REGION Network 10: Pulsing temperature and pressure same
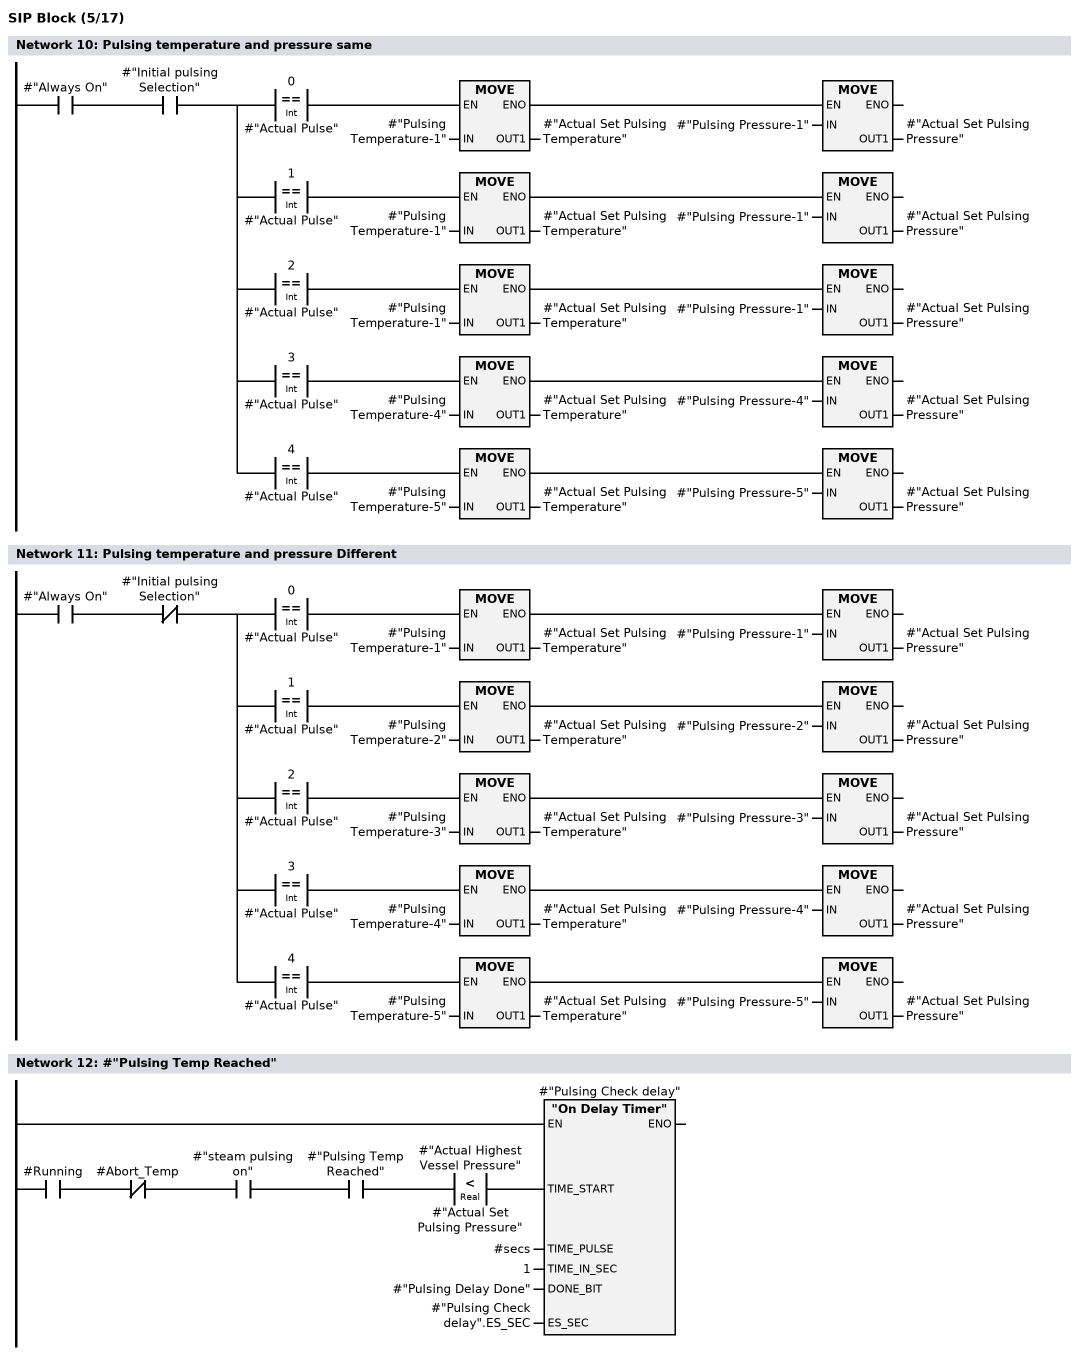
   RUNG wire#powerrail
      Contact( #"Always On" )
      Contact( #"Initial pulsing Selection" )
      wire#w1
      { S7_Templates := "SrcType := Int" } EQ_Contact(in1 := 0, in2 := #"Actual Pulse")
      Move(in := #"Pulsing Temperature-1", out1 => #"Actual Set Pulsing Temperature")
      Move(in := #"Pulsing Pressure-1", out1 => #"Actual Set Pulsing Pressure")
   END_RUNG
   RUNG wire#w1
      { S7_Templates := "SrcType := Int" } EQ_Contact(in1 := 1, in2 := #"Actual Pulse")
      Move(in := #"Pulsing Temperature-1", out1 => #"Actual Set Pulsing Temperature")
      Move(in := #"Pulsing Pressure-1", out1 => #"Actual Set Pulsing Pressure")
   END_RUNG
   RUNG wire#w1
      { S7_Templates := "SrcType := Int" } EQ_Contact(in1 := 2, in2 := #"Actual Pulse")
      Move(in := #"Pulsing Temperature-1", out1 => #"Actual Set Pulsing Temperature")
      Move(in := #"Pulsing Pressure-1", out1 => #"Actual Set Pulsing Pressure")
   END_RUNG
   RUNG wire#w1
      { S7_Templates := "SrcType := Int" } EQ_Contact(in1 := 3, in2 := #"Actual Pulse")
      Move(in := #"Pulsing Temperature-4", out1 => #"Actual Set Pulsing Temperature")
      Move(in := #"Pulsing Pressure-4", out1 => #"Actual Set Pulsing Pressure")
   END_RUNG
   RUNG wire#w1
      { S7_Templates := "SrcType := Int" } EQ_Contact(in1 := 4, in2 := #"Actual Pulse")
      Move(in := #"Pulsing Temperature-5", out1 => #"Actual Set Pulsing Temperature")
      Move(in := #"Pulsing Pressure-5", out1 => #"Actual Set Pulsing Pressure")
   END_RUNG
   // the same network as SCL:
   #_w1 := #"Always On" AND #"Initial pulsing Selection";
   IF #_w1 AND (0 = #"Actual Pulse") THEN
       #"Actual Set Pulsing Temperature" := #"Pulsing Temperature-1";
       #"Actual Set Pulsing Pressure" := #"Pulsing Pressure-1";
   END_IF;
   IF #_w1 AND (1 = #"Actual Pulse") THEN
       #"Actual Set Pulsing Temperature" := #"Pulsing Temperature-1";
       #"Actual Set Pulsing Pressure" := #"Pulsing Pressure-1";
   END_IF;
   IF #_w1 AND (2 = #"Actual Pulse") THEN
       #"Actual Set Pulsing Temperature" := #"Pulsing Temperature-1";
       #"Actual Set Pulsing Pressure" := #"Pulsing Pressure-1";
   END_IF;
   IF #_w1 AND (3 = #"Actual Pulse") THEN
       #"Actual Set Pulsing Temperature" := #"Pulsing Temperature-4";
       #"Actual Set Pulsing Pressure" := #"Pulsing Pressure-4";
   END_IF;
   IF #_w1 AND (4 = #"Actual Pulse") THEN
       #"Actual Set Pulsing Temperature" := #"Pulsing Temperature-5";
       #"Actual Set Pulsing Pressure" := #"Pulsing Pressure-5";
   END_IF;
END_REGION

REGION Network 11: Pulsing temperature and pressure Different
   RUNG wire#powerrail
      Contact( #"Always On" )
      I_Contact( #"Initial pulsing Selection" )
      wire#w1
      { S7_Templates := "SrcType := Int" } EQ_Contact(in1 := 0, in2 := #"Actual Pulse")
      Move(in := #"Pulsing Temperature-1", out1 => #"Actual Set Pulsing Temperature")
      Move(in := #"Pulsing Pressure-1", out1 => #"Actual Set Pulsing Pressure")
   END_RUNG
   RUNG wire#w1
      { S7_Templates := "SrcType := Int" } EQ_Contact(in1 := 1, in2 := #"Actual Pulse")
      Move(in := #"Pulsing Temperature-2", out1 => #"Actual Set Pulsing Temperature")
      Move(in := #"Pulsing Pressure-2", out1 => #"Actual Set Pulsing Pressure")
   END_RUNG
   RUNG wire#w1
      { S7_Templates := "SrcType := Int" } EQ_Contact(in1 := 2, in2 := #"Actual Pulse")
      Move(in := #"Pulsing Temperature-3", out1 => #"Actual Set Pulsing Temperature")
      Move(in := #"Pulsing Pressure-3", out1 => #"Actual Set Pulsing Pressure")
   END_RUNG
   RUNG wire#w1
      { S7_Templates := "SrcType := Int" } EQ_Contact(in1 := 3, in2 := #"Actual Pulse")
      Move(in := #"Pulsing Temperature-4", out1 => #"Actual Set Pulsing Temperature")
      Move(in := #"Pulsing Pressure-4", out1 => #"Actual Set Pulsing Pressure")
   END_RUNG
   RUNG wire#w1
      { S7_Templates := "SrcType := Int" } EQ_Contact(in1 := 4, in2 := #"Actual Pulse")
      Move(in := #"Pulsing Temperature-5", out1 => #"Actual Set Pulsing Temperature")
      Move(in := #"Pulsing Pressure-5", out1 => #"Actual Set Pulsing Pressure")
   END_RUNG
   // the same network as SCL:
   #_w1 := #"Always On" AND NOT #"Initial pulsing Selection";
   IF #_w1 AND (0 = #"Actual Pulse") THEN
       #"Actual Set Pulsing Temperature" := #"Pulsing Temperature-1";
       #"Actual Set Pulsing Pressure" := #"Pulsing Pressure-1";
   END_IF;
   IF #_w1 AND (1 = #"Actual Pulse") THEN
       #"Actual Set Pulsing Temperature" := #"Pulsing Temperature-2";
       #"Actual Set Pulsing Pressure" := #"Pulsing Pressure-2";
   END_IF;
   IF #_w1 AND (2 = #"Actual Pulse") THEN
       #"Actual Set Pulsing Temperature" := #"Pulsing Temperature-3";
       #"Actual Set Pulsing Pressure" := #"Pulsing Pressure-3";
   END_IF;
   IF #_w1 AND (3 = #"Actual Pulse") THEN
       #"Actual Set Pulsing Temperature" := #"Pulsing Temperature-4";
       #"Actual Set Pulsing Pressure" := #"Pulsing Pressure-4";
   END_IF;
   IF #_w1 AND (4 = #"Actual Pulse") THEN
       #"Actual Set Pulsing Temperature" := #"Pulsing Temperature-5";
       #"Actual Set Pulsing Pressure" := #"Pulsing Pressure-5";
   END_IF;
END_REGION

REGION Network 12: #"Pulsing Temp Reached"
   RUNG wire#powerrail
      #"Pulsing Check delay"(TIME_START := wire#w1, TIME_PULSE := #secs, TIME_IN_SEC := 1, DONE_BIT := #"Pulsing Delay Done", ES_SEC := #"Pulsing Check delay".ES_SEC)
   END_RUNG
   RUNG wire#powerrail
      Contact( #Running )
      I_Contact( #Abort_Temp )
      Contact( #"steam pulsing on" )
      Contact( #"Pulsing Temp Reached" )
      { S7_Templates := "SrcType := Real" } LT_Contact(in1 := #"Actual Highest Vessel Pressure", in2 := #"Actual Set Pulsing Pressure")
   END_RUNG wire#w1
   // the same network as SCL:
   #"Pulsing Check delay"(TIME_START := #Running AND NOT #Abort_Temp AND #"steam pulsing on" AND #"Pulsing Temp Reached" AND (#"Actual Highest Vessel Pressure" < #"Actual Set Pulsing Pressure"),   // "On Delay Timer"
                          TIME_PULSE := #secs,
                          TIME_IN_SEC := 1,
                          DONE_BIT := #"Pulsing Delay Done",
                          ES_SEC := #"Pulsing Check delay".ES_SEC);
END_REGION

REGION Network 13: #"Pulsing Temp Reached"
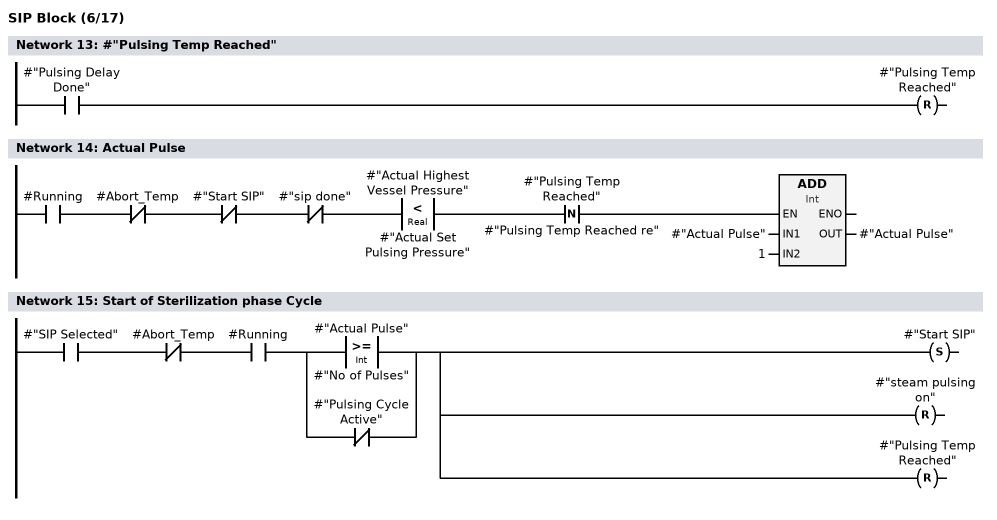
   RUNG wire#powerrail
      Contact( #"Pulsing Delay Done" )
      R_Coil( #"Pulsing Temp Reached" )
   END_RUNG
   // the same network as SCL:
   IF #"Pulsing Delay Done" THEN #"Pulsing Temp Reached" := FALSE; END_IF;
END_REGION

REGION Network 14: Actual Pulse
   RUNG wire#powerrail
      Contact( #Running )
      I_Contact( #Abort_Temp )
      I_Contact( #"Start SIP" )
      I_Contact( #"sip done" )
      { S7_Templates := "SrcType := Real" } LT_Contact(in1 := #"Actual Highest Vessel Pressure", in2 := #"Actual Set Pulsing Pressure")
      N_Contact(operand := #"Pulsing Temp Reached", bit := #"Pulsing Temp Reached re")
      { S7_Templates := "SrcType := Int"; S7_GenerateENO := "TRUE" } Add(in1 := #"Actual Pulse", in2 := 1, out => #"Actual Pulse")
   END_RUNG
   // the same network as SCL:
   #_w1 := #Running AND NOT #Abort_Temp AND NOT #"Start SIP" AND NOT #"sip done" AND (#"Actual Highest Vessel Pressure" < #"Actual Set Pulsing Pressure") AND NOT #"Pulsing Temp Reached" AND #"Pulsing Temp Reached re";   // falling edge of #"Pulsing Temp Reached"
   #"Pulsing Temp Reached re" := #"Pulsing Temp Reached";
   IF #_w1 THEN #"Actual Pulse" := #"Actual Pulse" + 1; END_IF;
END_REGION

REGION Network 15: Start of Sterilization phase Cycle
   RUNG wire#powerrail
      Contact( #"SIP Selected" )
      I_Contact( #Abort_Temp )
      Contact( #Running )
      wire#w1
      { S7_Templates := "SrcType := Int" } GE_Contact(in1 := #"Actual Pulse", in2 := #"No of Pulses")
      wire#w2
      S_Coil( #"Start SIP" )
   END_RUNG
   RUNG wire#w1
      I_Contact( #"Pulsing Cycle Active" )
   END_RUNG wire#w2
   RUNG wire#w2
      R_Coil( #"steam pulsing on" )
   END_RUNG
   RUNG wire#w2
      R_Coil( #"Pulsing Temp Reached" )
   END_RUNG
   // the same network as SCL:
   IF #"SIP Selected" AND NOT #Abort_Temp AND #Running AND ((#"Actual Pulse" >= #"No of Pulses") OR NOT #"Pulsing Cycle Active") THEN
       #"Start SIP" := TRUE;
       #"steam pulsing on" := FALSE;
       #"Pulsing Temp Reached" := FALSE;
   END_IF;
END_REGION

REGION Network 16: SIP Logic
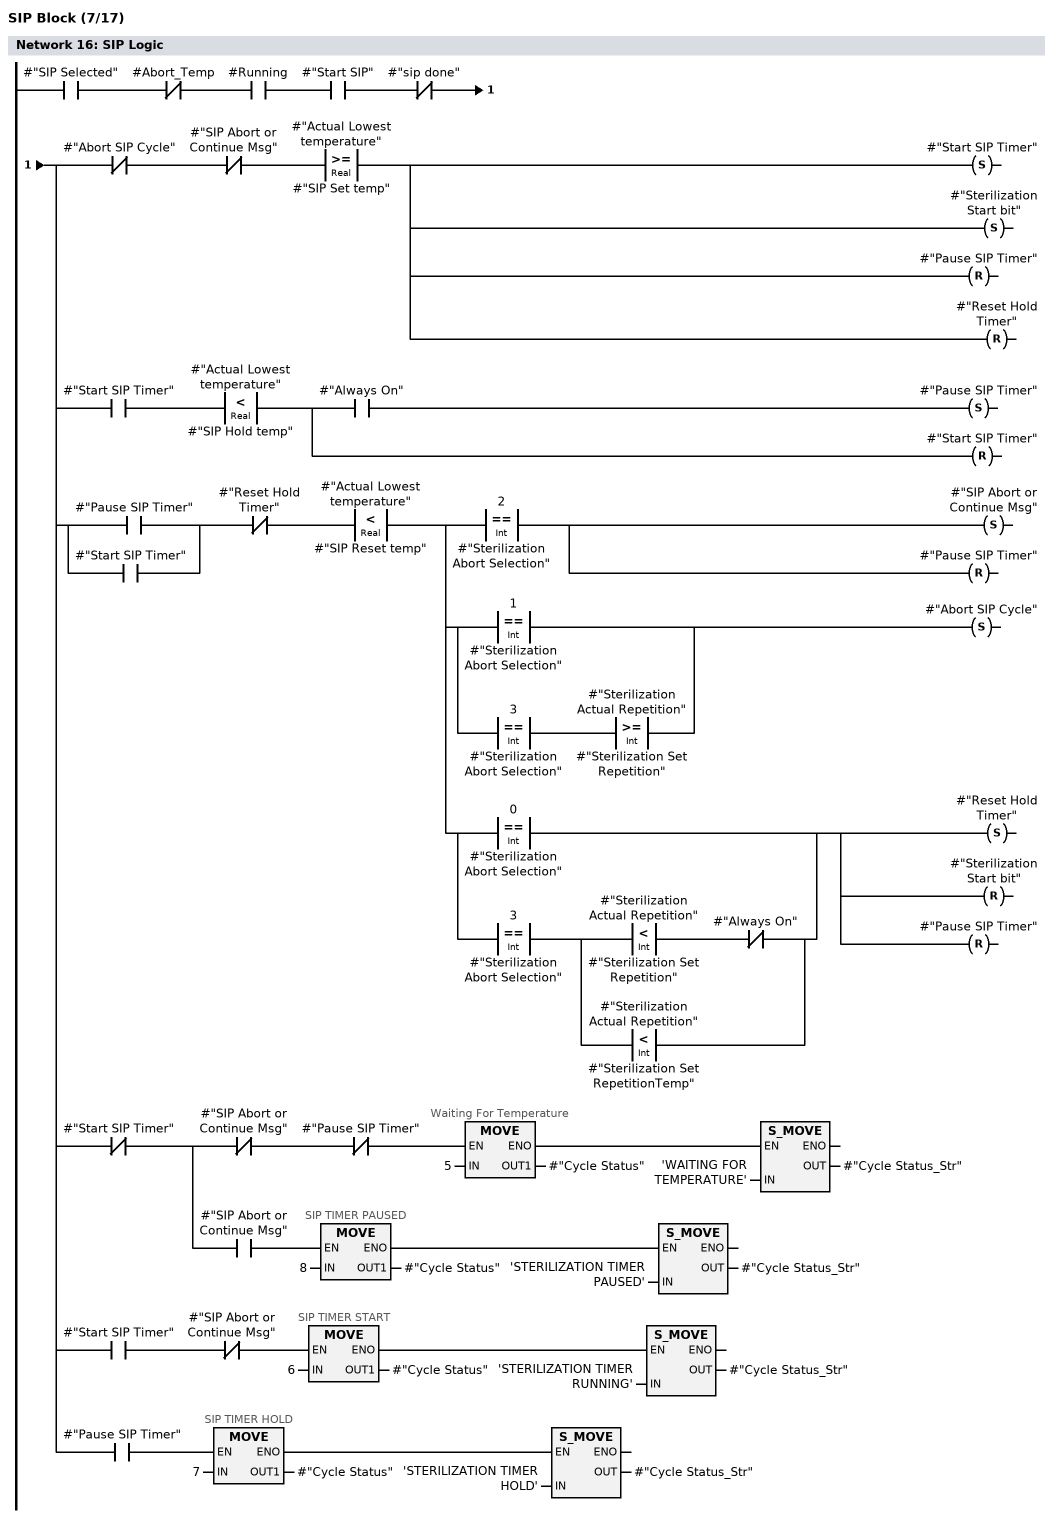
   RUNG wire#powerrail
      Contact( #"SIP Selected" )
      I_Contact( #Abort_Temp )
      Contact( #Running )
      Contact( #"Start SIP" )
      I_Contact( #"sip done" )
      wire#w1
      I_Contact( #"Abort SIP Cycle" )
      I_Contact( #"SIP Abort or Continue Msg" )
      { S7_Templates := "SrcType := Real" } GE_Contact(in1 := #"Actual Lowest temperature", in2 := #"SIP Set temp")
      wire#w2
      S_Coil( #"Start SIP Timer" )
   END_RUNG
   RUNG wire#w2
      S_Coil( #"Sterilization Start bit" )
   END_RUNG
   RUNG wire#w2
      R_Coil( #"Pause SIP Timer" )
   END_RUNG
   RUNG wire#w2
      R_Coil( #"Reset Hold Timer" )
   END_RUNG
   RUNG wire#w1
      Contact( #"Start SIP Timer" )
      { S7_Templates := "SrcType := Real" } LT_Contact(in1 := #"Actual Lowest temperature", in2 := #"SIP Hold temp")
      wire#w3
      Contact( #"Always On" )
      S_Coil( #"Pause SIP Timer" )
   END_RUNG
   RUNG wire#w3
      R_Coil( #"Start SIP Timer" )
   END_RUNG
   RUNG wire#w1
      Contact( #"Pause SIP Timer" )
      wire#w4
      I_Contact( #"Reset Hold Timer" )
      { S7_Templates := "SrcType := Real" } LT_Contact(in1 := #"Actual Lowest temperature", in2 := #"SIP Reset temp")
      wire#w5
      { S7_Templates := "SrcType := Int" } EQ_Contact(in1 := 2, in2 := #"Sterilization Abort Selection")
      wire#w6
      S_Coil( #"SIP Abort or Continue Msg" )
   END_RUNG
   RUNG wire#w1
      Contact( #"Start SIP Timer" )
   END_RUNG wire#w4
   RUNG wire#w6
      R_Coil( #"Pause SIP Timer" )
   END_RUNG
   RUNG wire#w5
      { S7_Templates := "SrcType := Int" } EQ_Contact(in1 := 1, in2 := #"Sterilization Abort Selection")
      wire#w7
      S_Coil( #"Abort SIP Cycle" )
   END_RUNG
   RUNG wire#w5
      { S7_Templates := "SrcType := Int" } EQ_Contact(in1 := 3, in2 := #"Sterilization Abort Selection")
      { S7_Templates := "SrcType := Int" } GE_Contact(in1 := #"Sterilization Actual Repetition", in2 := #"Sterilization Set Repetition")
   END_RUNG wire#w7
   RUNG wire#w5
      { S7_Templates := "SrcType := Int" } EQ_Contact(in1 := 0, in2 := #"Sterilization Abort Selection")
      wire#w8
      S_Coil( #"Reset Hold Timer" )
   END_RUNG
   RUNG wire#w5
      { S7_Templates := "SrcType := Int" } EQ_Contact(in1 := 3, in2 := #"Sterilization Abort Selection")
      wire#w9
      { S7_Templates := "SrcType := Int" } LT_Contact(in1 := #"Sterilization Actual Repetition", in2 := #"Sterilization Set Repetition")
      I_Contact( #"Always On" )
   END_RUNG wire#w8
   RUNG wire#w9
      { S7_Templates := "SrcType := Int" } LT_Contact(in1 := #"Sterilization Actual Repetition", in2 := #"Sterilization Set RepetitionTemp")
   END_RUNG wire#w8
   RUNG wire#w8
      R_Coil( #"Sterilization Start bit" )
   END_RUNG
   RUNG wire#w8
      R_Coil( #"Pause SIP Timer" )
   END_RUNG
   RUNG wire#w1
      I_Contact( #"Start SIP Timer" )
      wire#w10
      I_Contact( #"SIP Abort or Continue Msg" )
      I_Contact( #"Pause SIP Timer" )
      { S7_GenerateENO := "TRUE" } Move(in := 5, out1 => #"Cycle Status")   // Waiting For Temperature
      S_Move(in := 'WAITING FOR TEMPERATURE', out => #"Cycle Status_Str")
   END_RUNG
   RUNG wire#w10
      Contact( #"SIP Abort or Continue Msg" )
      { S7_GenerateENO := "TRUE" } Move(in := 8, out1 => #"Cycle Status")   // SIP TIMER PAUSED
      S_Move(in := 'STERILIZATION TIMER PAUSED', out => #"Cycle Status_Str")
   END_RUNG
   RUNG wire#w1
      Contact( #"Start SIP Timer" )
      I_Contact( #"SIP Abort or Continue Msg" )
      { S7_GenerateENO := "TRUE" } Move(in := 6, out1 => #"Cycle Status")   // SIP TIMER START
      S_Move(in := 'STERILIZATION TIMER RUNNING', out => #"Cycle Status_Str")
   END_RUNG
   RUNG wire#w1
      Contact( #"Pause SIP Timer" )
      { S7_GenerateENO := "TRUE" } Move(in := 7, out1 => #"Cycle Status")   // SIP TIMER HOLD
      S_Move(in := 'STERILIZATION TIMER HOLD', out => #"Cycle Status_Str")
   END_RUNG
   // the same network as SCL:
   // ENO of a box is taken as its EN; it also drops when the box reports an error
   #_w1 := #"SIP Selected" AND NOT #Abort_Temp AND #Running AND #"Start SIP" AND NOT #"sip done";
   IF #_w1 AND NOT #"Abort SIP Cycle" AND NOT #"SIP Abort or Continue Msg" AND (#"Actual Lowest temperature" >= #"SIP Set temp") THEN
       #"Start SIP Timer" := TRUE;
       #"Sterilization Start bit" := TRUE;
       #"Pause SIP Timer" := FALSE;
       #"Reset Hold Timer" := FALSE;
   END_IF;
   #_w2 := #_w1 AND #"Start SIP Timer" AND (#"Actual Lowest temperature" < #"SIP Hold temp");
   IF #_w2 AND #"Always On" THEN #"Pause SIP Timer" := TRUE; END_IF;
   IF #_w2 THEN #"Start SIP Timer" := FALSE; END_IF;
   #_w3 := #_w1 AND (#"Pause SIP Timer" OR #"Start SIP Timer") AND NOT #"Reset Hold Timer" AND (#"Actual Lowest temperature" < #"SIP Reset temp");
   IF #_w3 AND (2 = #"Sterilization Abort Selection") THEN
       #"SIP Abort or Continue Msg" := TRUE;
       #"Pause SIP Timer" := FALSE;
   END_IF;
   IF #_w3 AND ((1 = #"Sterilization Abort Selection") OR ((3 = #"Sterilization Abort Selection") AND (#"Sterilization Actual Repetition" >= #"Sterilization Set Repetition"))) THEN
       #"Abort SIP Cycle" := TRUE;
   END_IF;
   IF #_w3 AND ((0 = #"Sterilization Abort Selection") OR ((3 = #"Sterilization Abort Selection") AND (((#"Sterilization Actual Repetition" < #"Sterilization Set Repetition") AND NOT #"Always On") OR (#"Sterilization Actual Repetition" < #"Sterilization Set RepetitionTemp")))) THEN
       #"Reset Hold Timer" := TRUE;
       #"Sterilization Start bit" := FALSE;
       #"Pause SIP Timer" := FALSE;
   END_IF;
   #_w4 := #_w1 AND NOT #"Start SIP Timer";
   IF #_w4 AND NOT #"SIP Abort or Continue Msg" AND NOT #"Pause SIP Timer" THEN
       #"Cycle Status" := 5;   // Waiting For Temperature
       #"Cycle Status_Str" := 'WAITING FOR TEMPERATURE';
   END_IF;
   IF #_w4 AND #"SIP Abort or Continue Msg" THEN
       #"Cycle Status" := 8;   // SIP TIMER PAUSED
       #"Cycle Status_Str" := 'STERILIZATION TIMER PAUSED';
   END_IF;
   IF #_w1 AND #"Start SIP Timer" AND NOT #"SIP Abort or Continue Msg" THEN
       #"Cycle Status" := 6;   // SIP TIMER START
       #"Cycle Status_Str" := 'STERILIZATION TIMER RUNNING';
   END_IF;
   IF #_w1 AND #"Pause SIP Timer" THEN
       #"Cycle Status" := 7;   // SIP TIMER HOLD
       #"Cycle Status_Str" := 'STERILIZATION TIMER HOLD';
   END_IF;
END_REGION

REGION Network 17: Selection 2 :Abort msg conditions
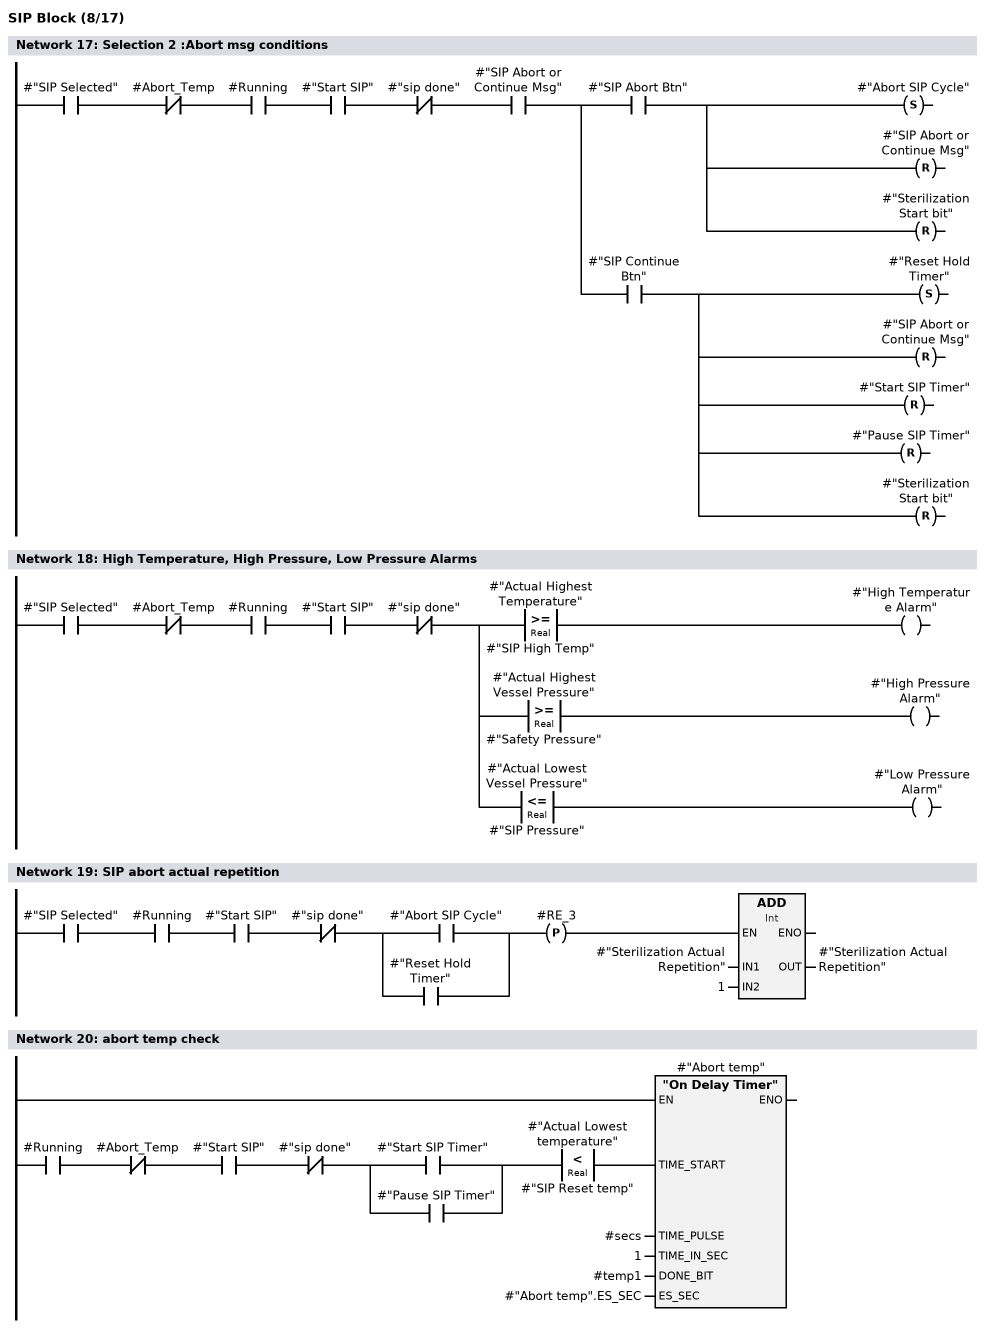
   RUNG wire#powerrail
      Contact( #"SIP Selected" )
      I_Contact( #Abort_Temp )
      Contact( #Running )
      Contact( #"Start SIP" )
      I_Contact( #"sip done" )
      Contact( #"SIP Abort or Continue Msg" )
      wire#w1
      Contact( #"SIP Abort Btn" )
      wire#w2
      S_Coil( #"Abort SIP Cycle" )
   END_RUNG
   RUNG wire#w2
      R_Coil( #"SIP Abort or Continue Msg" )
   END_RUNG
   RUNG wire#w2
      R_Coil( #"Sterilization Start bit" )
   END_RUNG
   RUNG wire#w1
      Contact( #"SIP Continue Btn" )
      wire#w3
      S_Coil( #"Reset Hold Timer" )
   END_RUNG
   RUNG wire#w3
      R_Coil( #"SIP Abort or Continue Msg" )
   END_RUNG
   RUNG wire#w3
      R_Coil( #"Start SIP Timer" )
   END_RUNG
   RUNG wire#w3
      R_Coil( #"Pause SIP Timer" )
   END_RUNG
   RUNG wire#w3
      R_Coil( #"Sterilization Start bit" )
   END_RUNG
   // the same network as SCL:
   #_w1 := #"SIP Selected" AND NOT #Abort_Temp AND #Running AND #"Start SIP" AND NOT #"sip done" AND #"SIP Abort or Continue Msg";
   IF #_w1 AND #"SIP Abort Btn" THEN
       #"Abort SIP Cycle" := TRUE;
       #"SIP Abort or Continue Msg" := FALSE;
       #"Sterilization Start bit" := FALSE;
   END_IF;
   IF #_w1 AND #"SIP Continue Btn" THEN
       #"Reset Hold Timer" := TRUE;
       #"SIP Abort or Continue Msg" := FALSE;
       #"Start SIP Timer" := FALSE;
       #"Pause SIP Timer" := FALSE;
       #"Sterilization Start bit" := FALSE;
   END_IF;
END_REGION

REGION Network 18: High Temperature, High Pressure, Low Pressure Alarms
   RUNG wire#powerrail
      Contact( #"SIP Selected" )
      I_Contact( #Abort_Temp )
      Contact( #Running )
      Contact( #"Start SIP" )
      I_Contact( #"sip done" )
      wire#w1
      { S7_Templates := "SrcType := Real" } GE_Contact(in1 := #"Actual Highest Temperature", in2 := #"SIP High Temp")
      Coil( #"High Temperature Alarm" )
   END_RUNG
   RUNG wire#w1
      { S7_Templates := "SrcType := Real" } GE_Contact(in1 := #"Actual Highest Vessel Pressure", in2 := #"Safety Pressure")
      Coil( #"High Pressure Alarm" )
   END_RUNG
   RUNG wire#w1
      { S7_Templates := "SrcType := Real" } LE_Contact(in1 := #"Actual Lowest Vessel Pressure", in2 := #"SIP Pressure")
      Coil( #"Low Pressure Alarm" )
   END_RUNG
   // the same network as SCL:
   #_w1 := #"SIP Selected" AND NOT #Abort_Temp AND #Running AND #"Start SIP" AND NOT #"sip done";
   #"High Temperature Alarm" := #_w1 AND (#"Actual Highest Temperature" >= #"SIP High Temp");
   #"High Pressure Alarm" := #_w1 AND (#"Actual Highest Vessel Pressure" >= #"Safety Pressure");
   #"Low Pressure Alarm" := #_w1 AND (#"Actual Lowest Vessel Pressure" <= #"SIP Pressure");
END_REGION

REGION Network 19: SIP abort actual repetition
   RUNG wire#powerrail
      Contact( #"SIP Selected" )
      Contact( #Running )
      Contact( #"Start SIP" )
      I_Contact( #"sip done" )
      wire#w1
      Contact( #"Abort SIP Cycle" )
      wire#w2
      P_Trig( #RE_3 )
      { S7_Templates := "SrcType := Int" } Add(in1 := #"Sterilization Actual Repetition", in2 := 1, out => #"Sterilization Actual Repetition")
   END_RUNG
   RUNG wire#w1
      Contact( #"Reset Hold Timer" )
   END_RUNG wire#w2
   // the same network as SCL:
   #_w1 := #"SIP Selected" AND #Running AND #"Start SIP" AND NOT #"sip done" AND (#"Abort SIP Cycle" OR #"Reset Hold Timer");
   #_w2 := #_w1 AND NOT #RE_3;   // rising edge
   #RE_3 := #_w1;
   IF #_w2 THEN #"Sterilization Actual Repetition" := #"Sterilization Actual Repetition" + 1; END_IF;
END_REGION

REGION Network 20: abort temp check
   RUNG wire#powerrail
      #"Abort temp"(TIME_START := wire#w3, TIME_PULSE := #secs, TIME_IN_SEC := 1, DONE_BIT := #temp1, ES_SEC := #"Abort temp".ES_SEC)
   END_RUNG
   RUNG wire#powerrail
      Contact( #Running )
      I_Contact( #Abort_Temp )
      Contact( #"Start SIP" )
      I_Contact( #"sip done" )
      wire#w1
      Contact( #"Start SIP Timer" )
      wire#w2
      { S7_Templates := "SrcType := Real" } LT_Contact(in1 := #"Actual Lowest temperature", in2 := #"SIP Reset temp")
   END_RUNG wire#w3
   RUNG wire#w1
      Contact( #"Pause SIP Timer" )
   END_RUNG wire#w2
   // the same network as SCL:
   #"Abort temp"(TIME_START := #Running AND NOT #Abort_Temp AND #"Start SIP" AND NOT #"sip done" AND (#"Start SIP Timer" OR #"Pause SIP Timer") AND (#"Actual Lowest temperature" < #"SIP Reset temp"),   // "On Delay Timer"
                 TIME_PULSE := #secs,
                 TIME_IN_SEC := 1,
                 DONE_BIT := #temp1,
                 ES_SEC := #"Abort temp".ES_SEC);
END_REGION

REGION Network 21: sip hold timer
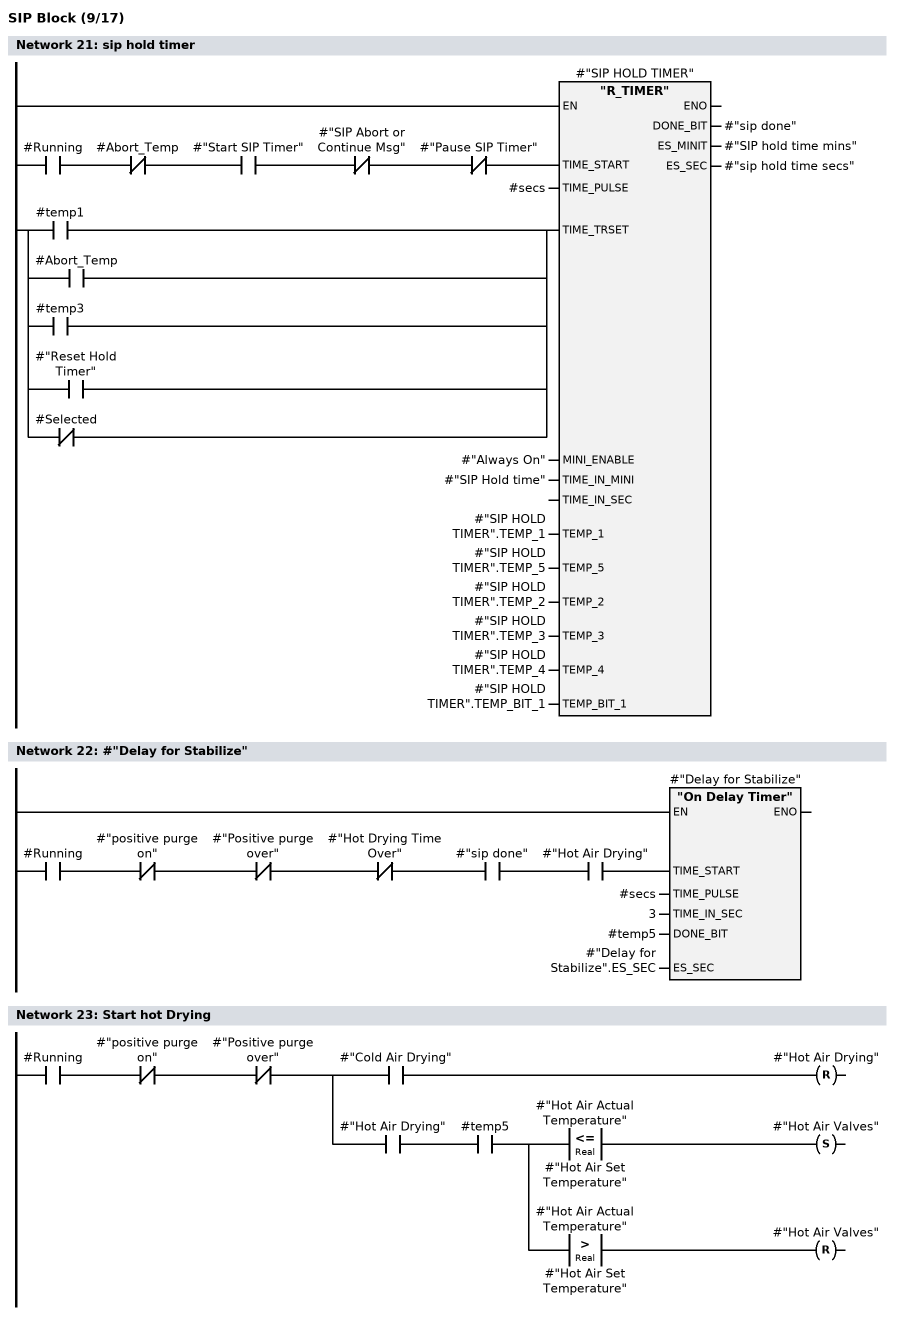
   RUNG wire#powerrail
      #"SIP HOLD TIMER"(TIME_START := wire#w1, TIME_TRSET := wire#w2, TIME_PULSE := #secs, MINI_ENABLE := #"Always On", TIME_IN_MINI := #"SIP Hold time", TIME_IN_SEC :=, TEMP_1 := #"SIP HOLD TIMER".TEMP_1, TEMP_5 := #"SIP HOLD TIMER".TEMP_5, TEMP_2 := #"SIP HOLD TIMER".TEMP_2, TEMP_3 := #"SIP HOLD TIMER".TEMP_3, TEMP_4 := #"SIP HOLD TIMER".TEMP_4, TEMP_BIT_1 := #"SIP HOLD TIMER".TEMP_BIT_1, DONE_BIT => #"sip done", ES_MINIT => #"SIP hold time mins", ES_SEC => #"sip hold time secs")
   END_RUNG
   RUNG wire#powerrail
      Contact( #Running )
      I_Contact( #Abort_Temp )
      Contact( #"Start SIP Timer" )
      I_Contact( #"SIP Abort or Continue Msg" )
      I_Contact( #"Pause SIP Timer" )
   END_RUNG wire#w1
   RUNG wire#powerrail
      Contact( #temp1 )
   END_RUNG wire#w2
   RUNG wire#powerrail
      Contact( #Abort_Temp )
   END_RUNG wire#w2
   RUNG wire#powerrail
      Contact( #temp3 )
   END_RUNG wire#w2
   RUNG wire#powerrail
      Contact( #"Reset Hold Timer" )
   END_RUNG wire#w2
   RUNG wire#powerrail
      I_Contact( #Selected )
   END_RUNG wire#w2
   // the same network as SCL:
   #"SIP HOLD TIMER"(TIME_START := #Running AND NOT #Abort_Temp AND #"Start SIP Timer" AND NOT #"SIP Abort or Continue Msg" AND NOT #"Pause SIP Timer",   // "R_TIMER"
                     TIME_PULSE := #secs,
                     TIME_TRSET := #temp1 OR #Abort_Temp OR #temp3 OR #"Reset Hold Timer" OR NOT #Selected,
                     MINI_ENABLE := #"Always On",
                     TIME_IN_MINI := #"SIP Hold time",
                     TEMP_1 := #"SIP HOLD TIMER".TEMP_1,
                     TEMP_5 := #"SIP HOLD TIMER".TEMP_5,
                     TEMP_2 := #"SIP HOLD TIMER".TEMP_2,
                     TEMP_3 := #"SIP HOLD TIMER".TEMP_3,
                     TEMP_4 := #"SIP HOLD TIMER".TEMP_4,
                     TEMP_BIT_1 := #"SIP HOLD TIMER".TEMP_BIT_1,
                     DONE_BIT => #"sip done",
                     ES_MINIT => #"SIP hold time mins",
                     ES_SEC => #"sip hold time secs");
END_REGION

REGION Network 22: #"Delay for Stabilize"
   RUNG wire#powerrail
      #"Delay for Stabilize"(TIME_START := wire#w1, TIME_PULSE := #secs, TIME_IN_SEC := 3, DONE_BIT := #temp5, ES_SEC := #"Delay for Stabilize".ES_SEC)
   END_RUNG
   RUNG wire#powerrail
      Contact( #Running )
      I_Contact( #"positive purge on" )
      I_Contact( #"Positive purge over" )
      I_Contact( #"Hot Drying Time Over" )
      Contact( #"sip done" )
      Contact( #"Hot Air Drying" )
   END_RUNG wire#w1
   // the same network as SCL:
   #"Delay for Stabilize"(TIME_START := #Running AND NOT #"positive purge on" AND NOT #"Positive purge over" AND NOT #"Hot Drying Time Over" AND #"sip done" AND #"Hot Air Drying",   // "On Delay Timer"
                          TIME_PULSE := #secs,
                          TIME_IN_SEC := 3,
                          DONE_BIT := #temp5,
                          ES_SEC := #"Delay for Stabilize".ES_SEC);
END_REGION

REGION Network 23: Start hot Drying
   RUNG wire#powerrail
      Contact( #Running )
      I_Contact( #"positive purge on" )
      I_Contact( #"Positive purge over" )
      wire#w1
      Contact( #"Cold Air Drying" )
      R_Coil( #"Hot Air Drying" )
   END_RUNG
   RUNG wire#w1
      Contact( #"Hot Air Drying" )
      Contact( #temp5 )
      wire#w2
      { S7_Templates := "SrcType := Real" } LE_Contact(in1 := #"Hot Air Actual Temperature", in2 := #"Hot Air Set Temperature")
      S_Coil( #"Hot Air Valves" )
   END_RUNG
   RUNG wire#w2
      { S7_Templates := "SrcType := Real" } GT_Contact(in1 := #"Hot Air Actual Temperature", in2 := #"Hot Air Set Temperature")
      R_Coil( #"Hot Air Valves" )
   END_RUNG
   // the same network as SCL:
   #_w1 := #Running AND NOT #"positive purge on" AND NOT #"Positive purge over";
   IF #_w1 AND #"Cold Air Drying" THEN #"Hot Air Drying" := FALSE; END_IF;
   #_w2 := #_w1 AND #"Hot Air Drying" AND #temp5;
   IF #_w2 AND (#"Hot Air Actual Temperature" <= #"Hot Air Set Temperature") THEN
       #"Hot Air Valves" := TRUE;
   END_IF;
   IF #_w2 AND (#"Hot Air Actual Temperature" > #"Hot Air Set Temperature") THEN
       #"Hot Air Valves" := FALSE;
   END_IF;
END_REGION

REGION Network 24: Hot Air Drying #"Actual Highest Vessel Pressure"
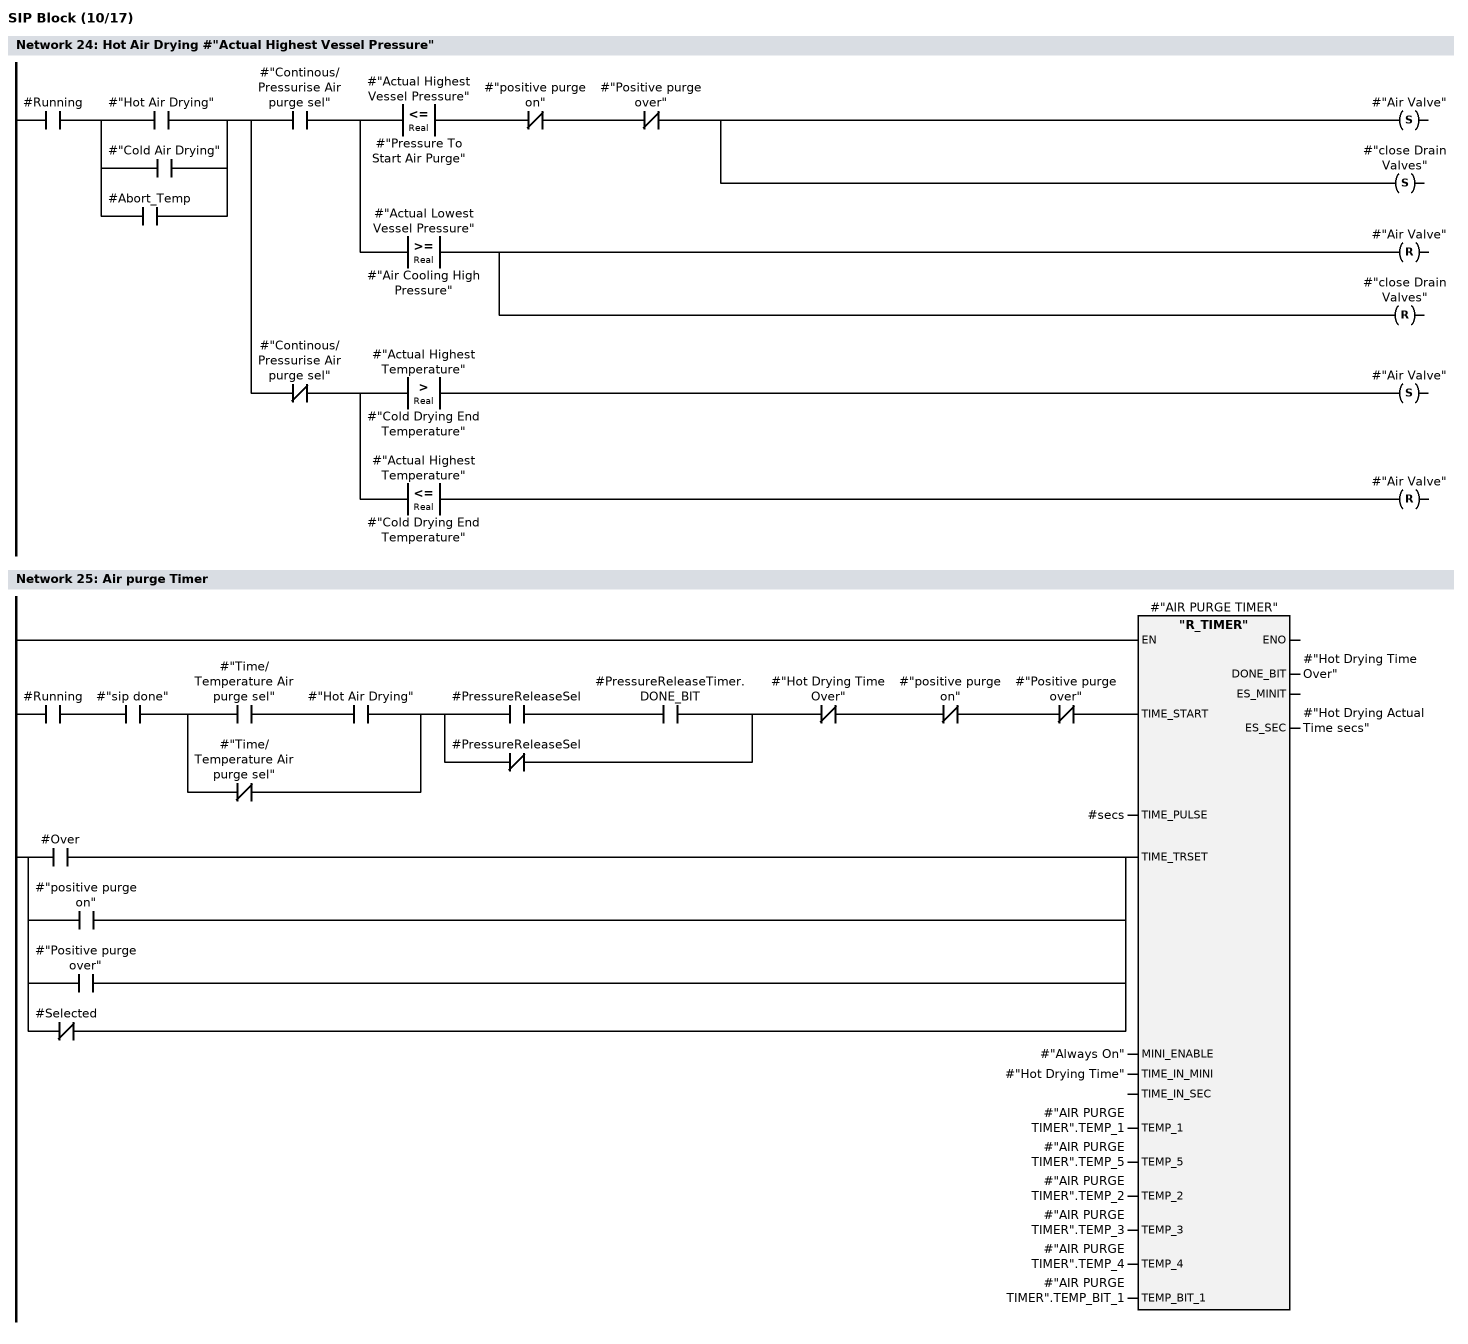
   RUNG wire#powerrail
      Contact( #Running )
      wire#w1
      Contact( #"Hot Air Drying" )
      wire#w2
      Contact( #"Continous/Pressurise Air purge sel" )
      wire#w3
      { S7_Templates := "SrcType := Real" } LE_Contact(in1 := #"Actual Highest Vessel Pressure", in2 := #"Pressure To Start Air Purge")
      I_Contact( #"positive purge on" )
      I_Contact( #"Positive purge over" )
      wire#w4
      S_Coil( #"Air Valve" )
   END_RUNG
   RUNG wire#w1
      Contact( #"Cold Air Drying" )
   END_RUNG wire#w2
   RUNG wire#w1
      Contact( #Abort_Temp )
   END_RUNG wire#w2
   RUNG wire#w4
      S_Coil( #"close Drain Valves" )
   END_RUNG
   RUNG wire#w3
      { S7_Templates := "SrcType := Real" } GE_Contact(in1 := #"Actual Lowest Vessel Pressure", in2 := #"Air Cooling High Pressure")
      wire#w5
      R_Coil( #"Air Valve" )
   END_RUNG
   RUNG wire#w5
      R_Coil( #"close Drain Valves" )
   END_RUNG
   RUNG wire#w2
      I_Contact( #"Continous/Pressurise Air purge sel" )
      wire#w6
      { S7_Templates := "SrcType := Real" } GT_Contact(in1 := #"Actual Highest Temperature", in2 := #"Cold Drying End Temperature")
      S_Coil( #"Air Valve" )
   END_RUNG
   RUNG wire#w6
      { S7_Templates := "SrcType := Real" } LE_Contact(in1 := #"Actual Highest Temperature", in2 := #"Cold Drying End Temperature")
      R_Coil( #"Air Valve" )
   END_RUNG
   // the same network as SCL:
   #_w1 := #Running AND (#"Hot Air Drying" OR #"Cold Air Drying" OR #Abort_Temp);
   #_w2 := #_w1 AND #"Continous/Pressurise Air purge sel";
   IF #_w2 AND (#"Actual Highest Vessel Pressure" <= #"Pressure To Start Air Purge") AND NOT #"positive purge on" AND NOT #"Positive purge over" THEN
       #"Air Valve" := TRUE;
       #"close Drain Valves" := TRUE;
   END_IF;
   IF #_w2 AND (#"Actual Lowest Vessel Pressure" >= #"Air Cooling High Pressure") THEN
       #"Air Valve" := FALSE;
       #"close Drain Valves" := FALSE;
   END_IF;
   #_w3 := #_w1 AND NOT #"Continous/Pressurise Air purge sel";
   IF #_w3 AND (#"Actual Highest Temperature" > #"Cold Drying End Temperature") THEN
       #"Air Valve" := TRUE;
   END_IF;
   IF #_w3 AND (#"Actual Highest Temperature" <= #"Cold Drying End Temperature") THEN
       #"Air Valve" := FALSE;
   END_IF;
END_REGION

REGION Network 25: Air purge Timer
   RUNG wire#powerrail
      #"AIR PURGE TIMER"(TIME_START := wire#w4, TIME_TRSET := wire#w5, TIME_PULSE := #secs, MINI_ENABLE := #"Always On", TIME_IN_MINI := #"Hot Drying Time", TIME_IN_SEC :=, TEMP_1 := #"AIR PURGE TIMER".TEMP_1, TEMP_5 := #"AIR PURGE TIMER".TEMP_5, TEMP_2 := #"AIR PURGE TIMER".TEMP_2, TEMP_3 := #"AIR PURGE TIMER".TEMP_3, TEMP_4 := #"AIR PURGE TIMER".TEMP_4, TEMP_BIT_1 := #"AIR PURGE TIMER".TEMP_BIT_1, DONE_BIT => #"Hot Drying Time Over", ES_MINIT =>, ES_SEC => #"Hot Drying Actual Time secs")
   END_RUNG
   RUNG wire#powerrail
      Contact( #Running )
      Contact( #"sip done" )
      wire#w1
      Contact( #"Time/Temperature Air purge sel" )
      Contact( #"Hot Air Drying" )
      wire#w2
      Contact( #PressureReleaseSel )
      Contact( #PressureReleaseTimer.DONE_BIT )
      wire#w3
      I_Contact( #"Hot Drying Time Over" )
      I_Contact( #"positive purge on" )
      I_Contact( #"Positive purge over" )
   END_RUNG wire#w4
   RUNG wire#w1
      I_Contact( #"Time/Temperature Air purge sel" )
   END_RUNG wire#w2
   RUNG wire#w2
      I_Contact( #PressureReleaseSel )
   END_RUNG wire#w3
   RUNG wire#powerrail
      Contact( #Over )
   END_RUNG wire#w5
   RUNG wire#powerrail
      Contact( #"positive purge on" )
   END_RUNG wire#w5
   RUNG wire#powerrail
      Contact( #"Positive purge over" )
   END_RUNG wire#w5
   RUNG wire#powerrail
      I_Contact( #Selected )
   END_RUNG wire#w5
   // the same network as SCL:
   #"AIR PURGE TIMER"(TIME_START := #Running AND #"sip done" AND ((#"Time/Temperature Air purge sel" AND #"Hot Air Drying") OR NOT #"Time/Temperature Air purge sel") AND ((#PressureReleaseSel AND #PressureReleaseTimer.DONE_BIT) OR NOT #PressureReleaseSel) AND NOT #"Hot Drying Time Over" AND NOT #"positive purge on" AND NOT #"Positive purge over",   // "R_TIMER"
                      TIME_PULSE := #secs,
                      TIME_TRSET := #Over OR #"positive purge on" OR #"Positive purge over" OR NOT #Selected,
                      MINI_ENABLE := #"Always On",
                      TIME_IN_MINI := #"Hot Drying Time",
                      TEMP_1 := #"AIR PURGE TIMER".TEMP_1,
                      TEMP_5 := #"AIR PURGE TIMER".TEMP_5,
                      TEMP_2 := #"AIR PURGE TIMER".TEMP_2,
                      TEMP_3 := #"AIR PURGE TIMER".TEMP_3,
                      TEMP_4 := #"AIR PURGE TIMER".TEMP_4,
                      TEMP_BIT_1 := #"AIR PURGE TIMER".TEMP_BIT_1,
                      DONE_BIT => #"Hot Drying Time Over",
                      ES_SEC => #"Hot Drying Actual Time secs");
END_REGION

REGION Network 26: Cold Air Drying
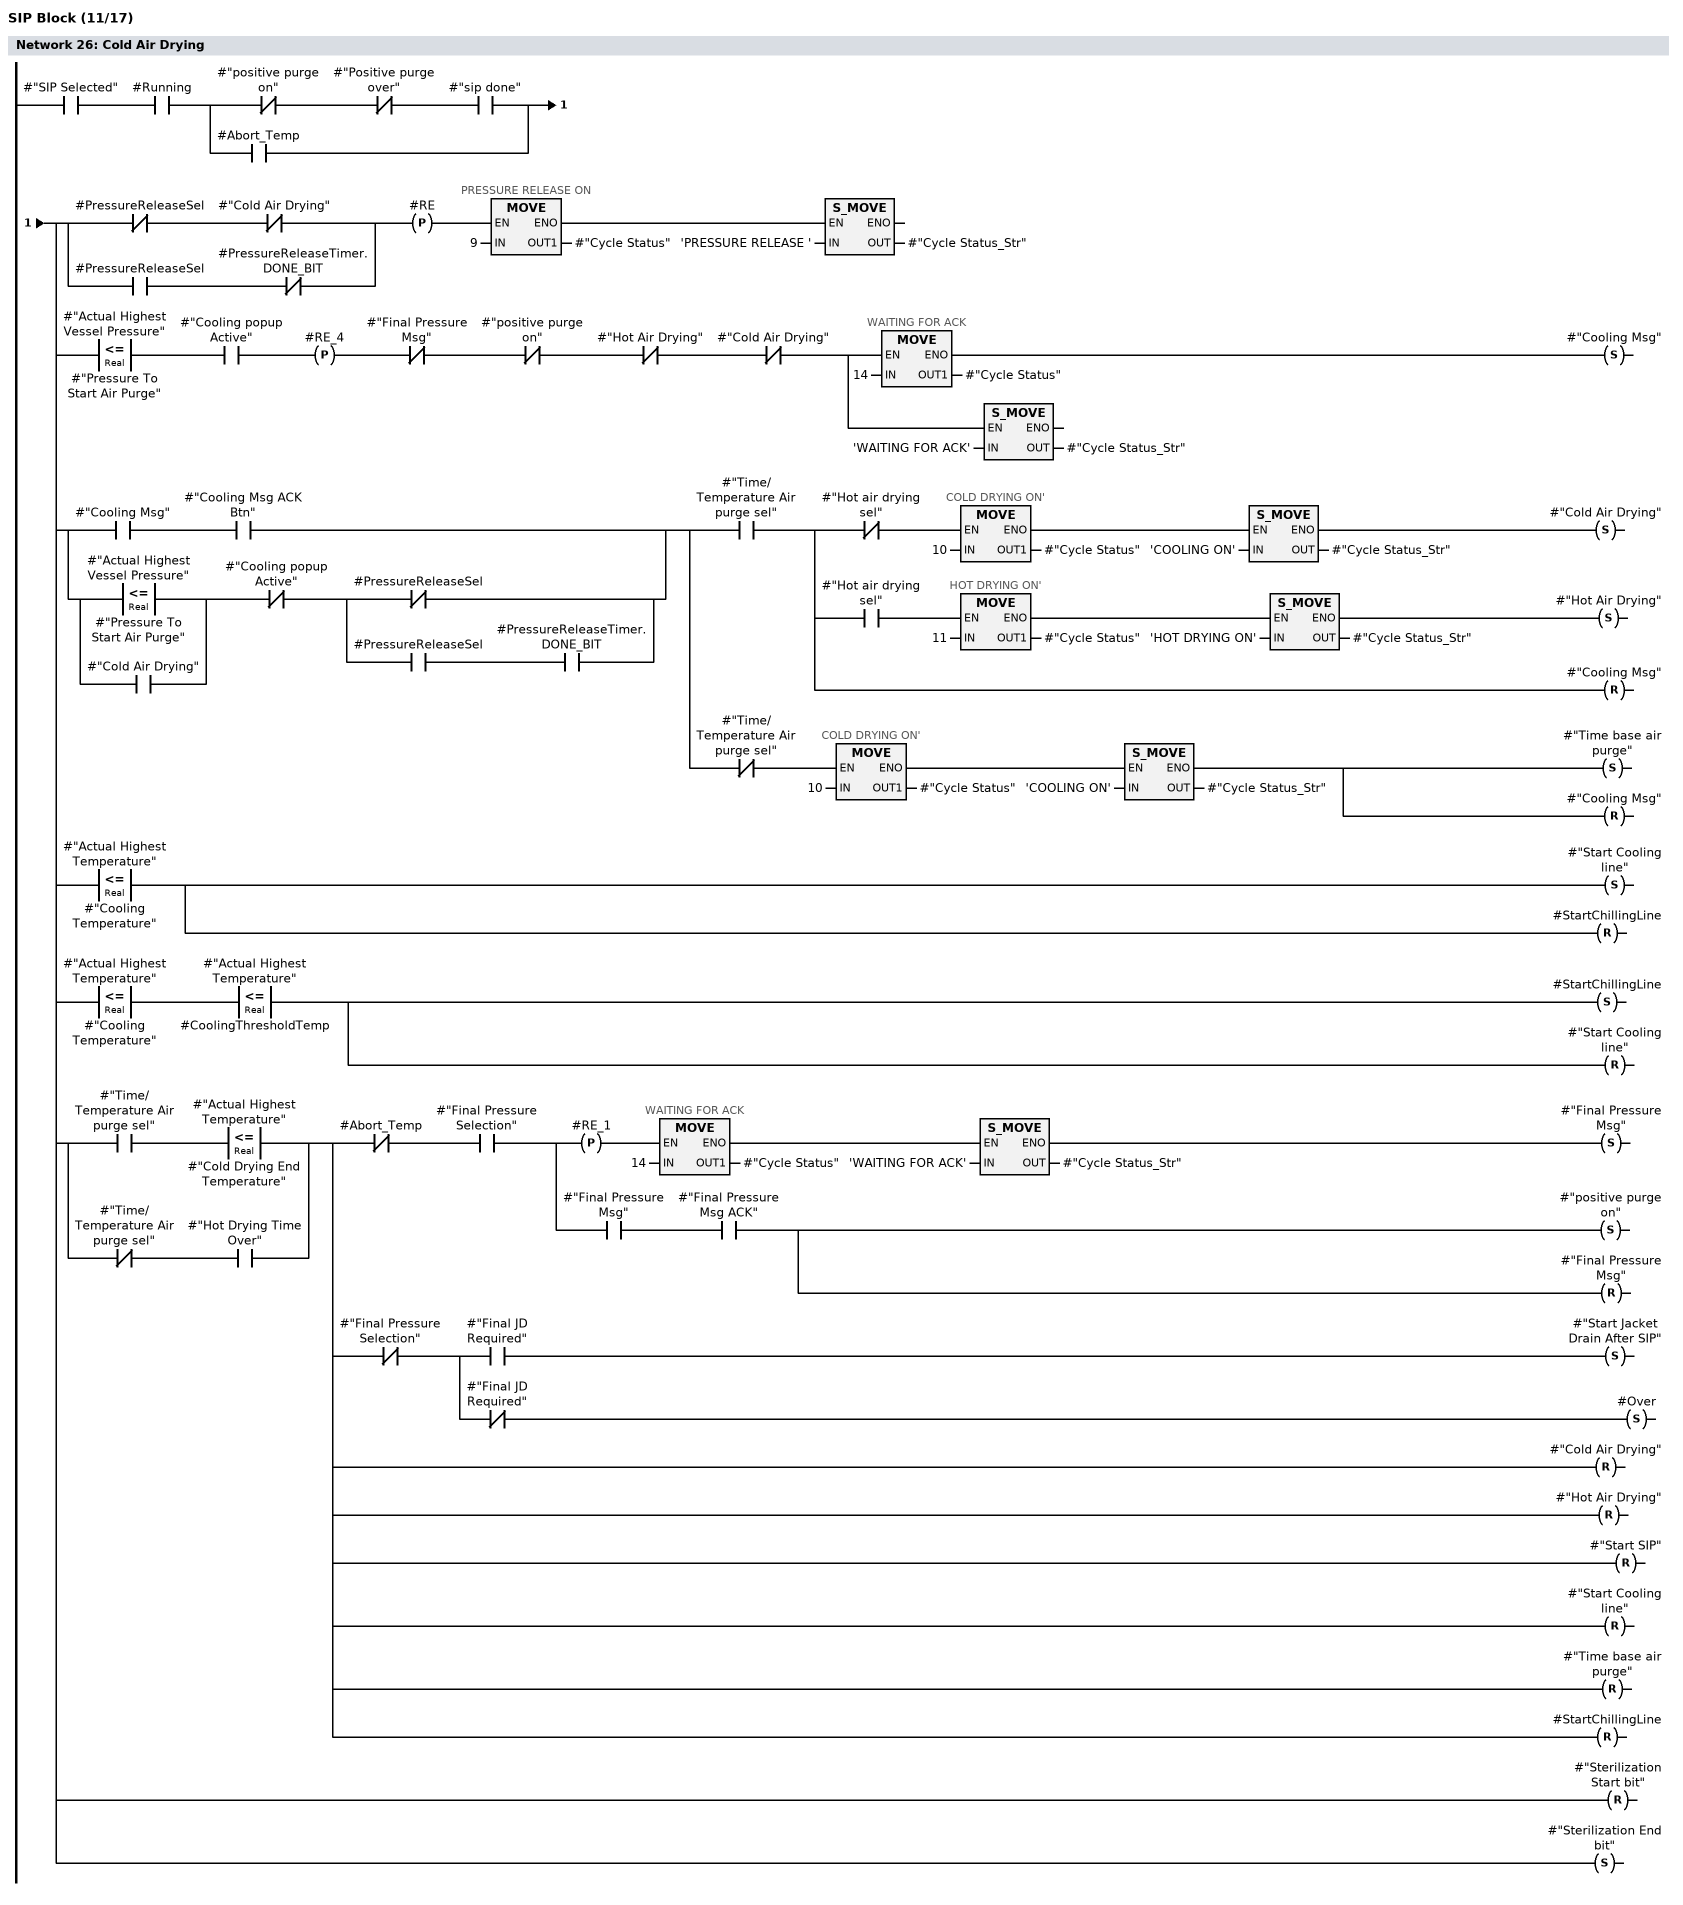
   RUNG wire#powerrail
      Contact( #"SIP Selected" )
      Contact( #Running )
      wire#w1
      I_Contact( #"positive purge on" )
      I_Contact( #"Positive purge over" )
      Contact( #"sip done" )
      wire#w2
      I_Contact( #PressureReleaseSel )
      I_Contact( #"Cold Air Drying" )
      wire#w3
      P_Trig( #RE )
      { S7_GenerateENO := "TRUE" } Move(in := 9, out1 => #"Cycle Status")   // PRESSURE RELEASE ON
      S_Move(in := 'PRESSURE RELEASE ', out => #"Cycle Status_Str")
   END_RUNG
   RUNG wire#w1
      Contact( #Abort_Temp )
   END_RUNG wire#w2
   RUNG wire#w2
      Contact( #PressureReleaseSel )
      I_Contact( #PressureReleaseTimer.DONE_BIT )
   END_RUNG wire#w3
   RUNG wire#w2
      { S7_Templates := "SrcType := Real" } LE_Contact(in1 := #"Actual Highest Vessel Pressure", in2 := #"Pressure To Start Air Purge")
      Contact( #"Cooling popup Active" )
      P_Trig( #RE_4 )
      I_Contact( #"Final Pressure Msg" )
      I_Contact( #"positive purge on" )
      I_Contact( #"Hot Air Drying" )
      I_Contact( #"Cold Air Drying" )
      wire#w4
      { S7_GenerateENO := "TRUE" } Move(in := 14, out1 => #"Cycle Status")   // WAITING FOR ACK
      S_Coil( #"Cooling Msg" )
   END_RUNG
   RUNG wire#w4
      S_Move(in := 'WAITING FOR ACK', out => #"Cycle Status_Str")
   END_RUNG
   RUNG wire#w2
      Contact( #"Cooling Msg" )
      Contact( #"Cooling Msg ACK Btn" )
      wire#w5
      Contact( #"Time/Temperature Air purge sel" )
      wire#w8
      I_Contact( #"Hot air drying sel" )
      { S7_GenerateENO := "TRUE" } Move(in := 10, out1 => #"Cycle Status")   // COLD DRYING ON'
      S_Move(in := 'COOLING ON', out => #"Cycle Status_Str")
      S_Coil( #"Cold Air Drying" )
   END_RUNG
   RUNG wire#w2
      { S7_Templates := "SrcType := Real" } LE_Contact(in1 := #"Actual Highest Vessel Pressure", in2 := #"Pressure To Start Air Purge")
      wire#w6
      I_Contact( #"Cooling popup Active" )
      wire#w7
      I_Contact( #PressureReleaseSel )
   END_RUNG wire#w5
   RUNG wire#w2
      Contact( #"Cold Air Drying" )
   END_RUNG wire#w6
   RUNG wire#w7
      Contact( #PressureReleaseSel )
      Contact( #PressureReleaseTimer.DONE_BIT )
   END_RUNG wire#w5
   RUNG wire#w8
      Contact( #"Hot air drying sel" )
      { S7_GenerateENO := "TRUE" } Move(in := 11, out1 => #"Cycle Status")   // HOT DRYING ON'
      S_Move(in := 'HOT DRYING ON', out => #"Cycle Status_Str")
      S_Coil( #"Hot Air Drying" )
   END_RUNG
   RUNG wire#w8
      R_Coil( #"Cooling Msg" )
   END_RUNG
   RUNG wire#w5
      I_Contact( #"Time/Temperature Air purge sel" )
      { S7_GenerateENO := "TRUE" } Move(in := 10, out1 => #"Cycle Status")   // COLD DRYING ON'
      S_Move(in := 'COOLING ON', out => #"Cycle Status_Str")
      wire#w9
      S_Coil( #"Time base air purge" )
   END_RUNG
   RUNG wire#w9
      R_Coil( #"Cooling Msg" )
   END_RUNG
   RUNG wire#w2
      { S7_Templates := "SrcType := Real" } LE_Contact(in1 := #"Actual Highest Temperature", in2 := #"Cooling Temperature")
      wire#w10
      S_Coil( #"Start Cooling line" )
   END_RUNG
   RUNG wire#w10
      R_Coil( #StartChillingLine )
   END_RUNG
   RUNG wire#w2
      { S7_Templates := "SrcType := Real" } LE_Contact(in1 := #"Actual Highest Temperature", in2 := #"Cooling Temperature")
      { S7_Templates := "SrcType := Real" } LE_Contact(in1 := #"Actual Highest Temperature", in2 := #CoolingThresholdTemp)
      wire#w11
      S_Coil( #StartChillingLine )
   END_RUNG
   RUNG wire#w11
      R_Coil( #"Start Cooling line" )
   END_RUNG
   RUNG wire#w2
      Contact( #"Time/Temperature Air purge sel" )
      { S7_Templates := "SrcType := Real" } LE_Contact(in1 := #"Actual Highest Temperature", in2 := #"Cold Drying End Temperature")
      wire#w12
      I_Contact( #Abort_Temp )
      Contact( #"Final Pressure Selection" )
      wire#w13
      P_Trig( #RE_1 )
      { S7_GenerateENO := "TRUE" } Move(in := 14, out1 => #"Cycle Status")   // WAITING FOR ACK
      S_Move(in := 'WAITING FOR ACK', out => #"Cycle Status_Str")
      S_Coil( #"Final Pressure Msg" )
   END_RUNG
   RUNG wire#w2
      I_Contact( #"Time/Temperature Air purge sel" )
      Contact( #"Hot Drying Time Over" )
   END_RUNG wire#w12
   RUNG wire#w13
      Contact( #"Final Pressure Msg" )
      Contact( #"Final Pressure Msg ACK" )
      wire#w14
      S_Coil( #"positive purge on" )
   END_RUNG
   RUNG wire#w14
      R_Coil( #"Final Pressure Msg" )
   END_RUNG
   RUNG wire#w12
      I_Contact( #"Final Pressure Selection" )
      wire#w15
      Contact( #"Final JD Required" )
      S_Coil( #"Start Jacket Drain After SIP" )
   END_RUNG
   RUNG wire#w15
      I_Contact( #"Final JD Required" )
      S_Coil( #Over )
   END_RUNG
   RUNG wire#w12
      R_Coil( #"Cold Air Drying" )
   END_RUNG
   RUNG wire#w12
      R_Coil( #"Hot Air Drying" )
   END_RUNG
   RUNG wire#w12
      R_Coil( #"Start SIP" )
   END_RUNG
   RUNG wire#w12
      R_Coil( #"Start Cooling line" )
   END_RUNG
   RUNG wire#w12
      R_Coil( #"Time base air purge" )
   END_RUNG
   RUNG wire#w12
      R_Coil( #StartChillingLine )
   END_RUNG
   RUNG wire#w2
      R_Coil( #"Sterilization Start bit" )
   END_RUNG
   RUNG wire#w2
      S_Coil( #"Sterilization End bit" )
   END_RUNG
   // the same network as SCL:
   // ENO of a box is taken as its EN; it also drops when the box reports an error
   #_w1 := #"SIP Selected" AND #Running AND ((NOT #"positive purge on" AND NOT #"Positive purge over" AND #"sip done") OR #Abort_Temp);
   #_w2 := #_w1 AND ((NOT #PressureReleaseSel AND NOT #"Cold Air Drying") OR (#PressureReleaseSel AND NOT #PressureReleaseTimer.DONE_BIT));
   #_w3 := #_w2 AND NOT #RE;   // rising edge
   #RE := #_w2;
   IF #_w3 THEN
       #"Cycle Status" := 9;   // PRESSURE RELEASE ON
       #"Cycle Status_Str" := 'PRESSURE RELEASE ';
   END_IF;
   #_w4 := #_w1 AND (#"Actual Highest Vessel Pressure" <= #"Pressure To Start Air Purge") AND #"Cooling popup Active";
   #_w5 := #_w4 AND NOT #RE_4;   // rising edge
   #RE_4 := #_w4;
   IF #_w5 AND NOT #"Final Pressure Msg" AND NOT #"positive purge on" AND NOT #"Hot Air Drying" AND NOT #"Cold Air Drying" THEN
       #"Cycle Status" := 14;   // WAITING FOR ACK
       #"Cooling Msg" := TRUE;
       #"Cycle Status_Str" := 'WAITING FOR ACK';
   END_IF;
   #_w6 := #_w1 AND ((#"Cooling Msg" AND #"Cooling Msg ACK Btn") OR (((#"Actual Highest Vessel Pressure" <= #"Pressure To Start Air Purge") OR #"Cold Air Drying") AND NOT #"Cooling popup Active" AND (NOT #PressureReleaseSel OR (#PressureReleaseSel AND #PressureReleaseTimer.DONE_BIT))));
   #_w7 := #_w6 AND #"Time/Temperature Air purge sel";
   IF #_w7 AND NOT #"Hot air drying sel" THEN
       #"Cycle Status" := 10;   // COLD DRYING ON'
       #"Cycle Status_Str" := 'COOLING ON';
       #"Cold Air Drying" := TRUE;
   END_IF;
   IF #_w7 AND #"Hot air drying sel" THEN
       #"Cycle Status" := 11;   // HOT DRYING ON'
       #"Cycle Status_Str" := 'HOT DRYING ON';
       #"Hot Air Drying" := TRUE;
   END_IF;
   IF #_w7 THEN #"Cooling Msg" := FALSE; END_IF;
   IF #_w6 AND NOT #"Time/Temperature Air purge sel" THEN
       #"Cycle Status" := 10;   // COLD DRYING ON'
       #"Cycle Status_Str" := 'COOLING ON';
       #"Time base air purge" := TRUE;
       #"Cooling Msg" := FALSE;
   END_IF;
   IF #_w1 AND (#"Actual Highest Temperature" <= #"Cooling Temperature") THEN
       #"Start Cooling line" := TRUE;
       #StartChillingLine := FALSE;
   END_IF;
   IF #_w1 AND (#"Actual Highest Temperature" <= #"Cooling Temperature") AND (#"Actual Highest Temperature" <= #CoolingThresholdTemp) THEN
       #StartChillingLine := TRUE;
       #"Start Cooling line" := FALSE;
   END_IF;
   #_w8 := #_w1 AND ((#"Time/Temperature Air purge sel" AND (#"Actual Highest Temperature" <= #"Cold Drying End Temperature")) OR (NOT #"Time/Temperature Air purge sel" AND #"Hot Drying Time Over"));
   #_w9 := #_w8 AND NOT #Abort_Temp AND #"Final Pressure Selection";
   #_w10 := #_w9 AND NOT #RE_1;   // rising edge
   #RE_1 := #_w9;
   IF #_w10 THEN
       #"Cycle Status" := 14;   // WAITING FOR ACK
       #"Cycle Status_Str" := 'WAITING FOR ACK';
       #"Final Pressure Msg" := TRUE;
   END_IF;
   IF #_w9 AND #"Final Pressure Msg" AND #"Final Pressure Msg ACK" THEN
       #"positive purge on" := TRUE;
       #"Final Pressure Msg" := FALSE;
   END_IF;
   #_w11 := #_w8 AND NOT #"Final Pressure Selection";
   IF #_w11 AND #"Final JD Required" THEN #"Start Jacket Drain After SIP" := TRUE; END_IF;
   IF #_w11 AND NOT #"Final JD Required" THEN #Over := TRUE; END_IF;
   IF #_w8 THEN
       #"Cold Air Drying" := FALSE;
       #"Hot Air Drying" := FALSE;
       #"Start SIP" := FALSE;
       #"Start Cooling line" := FALSE;
       #"Time base air purge" := FALSE;
       #StartChillingLine := FALSE;
   END_IF;
   IF #_w1 THEN
       #"Sterilization Start bit" := FALSE;
       #"Sterilization End bit" := TRUE;
   END_IF;
END_REGION

REGION Network 27: #"Hot Air Valves"
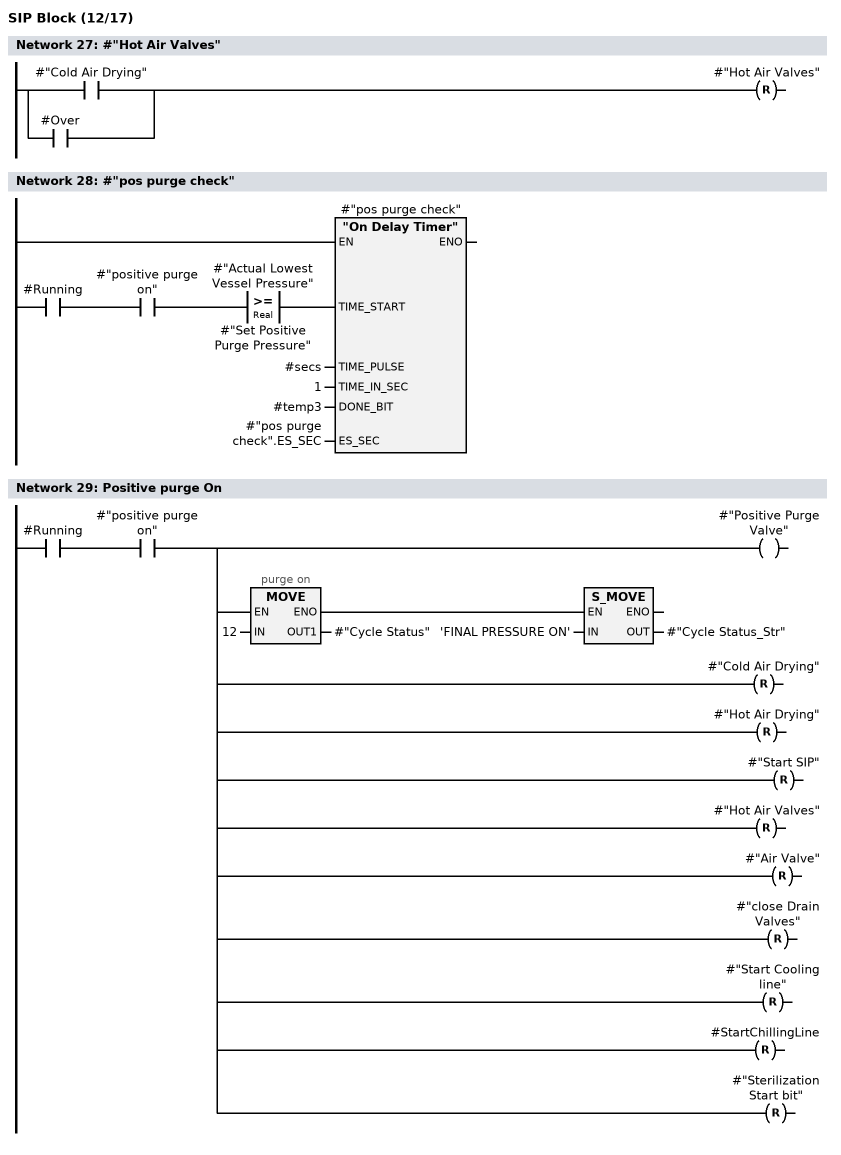
   RUNG wire#powerrail
      Contact( #"Cold Air Drying" )
      wire#w1
      R_Coil( #"Hot Air Valves" )
   END_RUNG
   RUNG wire#powerrail
      Contact( #Over )
   END_RUNG wire#w1
   // the same network as SCL:
   IF #"Cold Air Drying" OR #Over THEN #"Hot Air Valves" := FALSE; END_IF;
END_REGION

REGION Network 28: #"pos purge check"
   RUNG wire#powerrail
      #"pos purge check"(TIME_START := wire#w1, TIME_PULSE := #secs, TIME_IN_SEC := 1, DONE_BIT := #temp3, ES_SEC := #"pos purge check".ES_SEC)
   END_RUNG
   RUNG wire#powerrail
      Contact( #Running )
      Contact( #"positive purge on" )
      { S7_Templates := "SrcType := Real" } GE_Contact(in1 := #"Actual Lowest Vessel Pressure", in2 := #"Set Positive Purge Pressure")
   END_RUNG wire#w1
   // the same network as SCL:
   #"pos purge check"(TIME_START := #Running AND #"positive purge on" AND (#"Actual Lowest Vessel Pressure" >= #"Set Positive Purge Pressure"),   // "On Delay Timer"
                      TIME_PULSE := #secs,
                      TIME_IN_SEC := 1,
                      DONE_BIT := #temp3,
                      ES_SEC := #"pos purge check".ES_SEC);
END_REGION

REGION Network 29: Positive purge On
   RUNG wire#powerrail
      Contact( #Running )
      Contact( #"positive purge on" )
      wire#w1
      Coil( #"Positive Purge Valve" )
   END_RUNG
   RUNG wire#w1
      { S7_GenerateENO := "TRUE" } Move(in := 12, out1 => #"Cycle Status")   // purge on
      S_Move(in := 'FINAL PRESSURE ON', out => #"Cycle Status_Str")
   END_RUNG
   RUNG wire#w1
      R_Coil( #"Cold Air Drying" )
   END_RUNG
   RUNG wire#w1
      R_Coil( #"Hot Air Drying" )
   END_RUNG
   RUNG wire#w1
      R_Coil( #"Start SIP" )
   END_RUNG
   RUNG wire#w1
      R_Coil( #"Hot Air Valves" )
   END_RUNG
   RUNG wire#w1
      R_Coil( #"Air Valve" )
   END_RUNG
   RUNG wire#w1
      R_Coil( #"close Drain Valves" )
   END_RUNG
   RUNG wire#w1
      R_Coil( #"Start Cooling line" )
   END_RUNG
   RUNG wire#w1
      R_Coil( #StartChillingLine )
   END_RUNG
   RUNG wire#w1
      R_Coil( #"Sterilization Start bit" )
   END_RUNG
   // the same network as SCL:
   // ENO of a box is taken as its EN; it also drops when the box reports an error
   #"Positive Purge Valve" := #Running AND #"positive purge on";
   IF #"Positive Purge Valve" THEN
       #"Cycle Status" := 12;   // purge on
       #"Cycle Status_Str" := 'FINAL PRESSURE ON';
       #"Cold Air Drying" := FALSE;
       #"Hot Air Drying" := FALSE;
       #"Start SIP" := FALSE;
       #"Hot Air Valves" := FALSE;
       #"Air Valve" := FALSE;
       #"close Drain Valves" := FALSE;
       #"Start Cooling line" := FALSE;
       #StartChillingLine := FALSE;
       #"Sterilization Start bit" := FALSE;
   END_IF;
END_REGION

REGION Network 30: positive pressure over
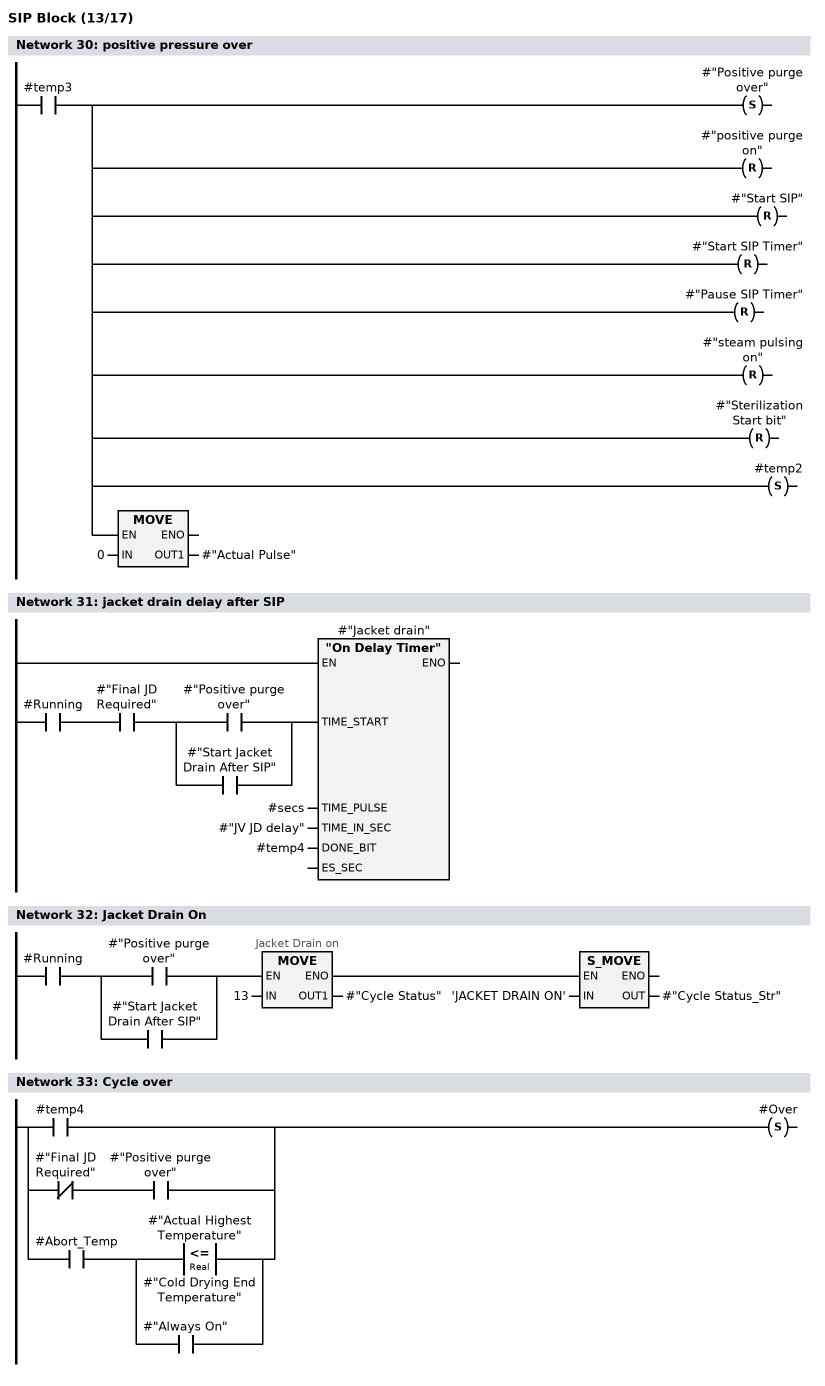
   RUNG wire#powerrail
      Contact( #temp3 )
      wire#w1
      S_Coil( #"Positive purge over" )
   END_RUNG
   RUNG wire#w1
      R_Coil( #"positive purge on" )
   END_RUNG
   RUNG wire#w1
      R_Coil( #"Start SIP" )
   END_RUNG
   RUNG wire#w1
      R_Coil( #"Start SIP Timer" )
   END_RUNG
   RUNG wire#w1
      R_Coil( #"Pause SIP Timer" )
   END_RUNG
   RUNG wire#w1
      R_Coil( #"steam pulsing on" )
   END_RUNG
   RUNG wire#w1
      R_Coil( #"Sterilization Start bit" )
   END_RUNG
   RUNG wire#w1
      S_Coil( #temp2 )
   END_RUNG
   RUNG wire#w1
      { S7_GenerateENO := "TRUE" } Move(in := 0, out1 => #"Actual Pulse")
   END_RUNG
   // the same network as SCL:
   IF #temp3 THEN
       #"Positive purge over" := TRUE;
       #"positive purge on" := FALSE;
       #"Start SIP" := FALSE;
       #"Start SIP Timer" := FALSE;
       #"Pause SIP Timer" := FALSE;
       #"steam pulsing on" := FALSE;
       #"Sterilization Start bit" := FALSE;
       #temp2 := TRUE;
       #"Actual Pulse" := 0;
   END_IF;
END_REGION

REGION Network 31: jacket drain delay after SIP
   RUNG wire#powerrail
      #"Jacket drain"(TIME_START := wire#w2, TIME_PULSE := #secs, TIME_IN_SEC := #"JV JD delay", DONE_BIT := #temp4, ES_SEC :=)
   END_RUNG
   RUNG wire#powerrail
      Contact( #Running )
      Contact( #"Final JD Required" )
      wire#w1
      Contact( #"Positive purge over" )
   END_RUNG wire#w2
   RUNG wire#w1
      Contact( #"Start Jacket Drain After SIP" )
   END_RUNG wire#w2
   // the same network as SCL:
   #"Jacket drain"(TIME_START := #Running AND #"Final JD Required" AND (#"Positive purge over" OR #"Start Jacket Drain After SIP"),   // "On Delay Timer"
                   TIME_PULSE := #secs,
                   TIME_IN_SEC := #"JV JD delay",
                   DONE_BIT := #temp4);
END_REGION

REGION Network 32: Jacket Drain On
   RUNG wire#powerrail
      Contact( #Running )
      wire#w1
      Contact( #"Positive purge over" )
      wire#w2
      { S7_GenerateENO := "TRUE" } Move(in := 13, out1 => #"Cycle Status")   // Jacket Drain on
      S_Move(in := 'JACKET DRAIN ON', out => #"Cycle Status_Str")
   END_RUNG
   RUNG wire#w1
      Contact( #"Start Jacket Drain After SIP" )
   END_RUNG wire#w2
   // the same network as SCL:
   // ENO of a box is taken as its EN; it also drops when the box reports an error
   IF #Running AND (#"Positive purge over" OR #"Start Jacket Drain After SIP") THEN
       #"Cycle Status" := 13;   // Jacket Drain on
       #"Cycle Status_Str" := 'JACKET DRAIN ON';
   END_IF;
END_REGION

REGION Network 33: Cycle over
   RUNG wire#powerrail
      Contact( #temp4 )
      wire#w1
      S_Coil( #Over )
   END_RUNG
   RUNG wire#powerrail
      I_Contact( #"Final JD Required" )
      Contact( #"Positive purge over" )
   END_RUNG wire#w1
   RUNG wire#powerrail
      Contact( #Abort_Temp )
      wire#w2
      { S7_Templates := "SrcType := Real" } LE_Contact(in1 := #"Actual Highest Temperature", in2 := #"Cold Drying End Temperature")
   END_RUNG wire#w1
   RUNG wire#w2
      Contact( #"Always On" )
   END_RUNG wire#w1
   // the same network as SCL:
   IF #temp4 OR (NOT #"Final JD Required" AND #"Positive purge over") OR (#Abort_Temp AND ((#"Actual Highest Temperature" <= #"Cold Drying End Temperature") OR #"Always On")) THEN
       #Over := TRUE;
   END_IF;
END_REGION

REGION Network 34: Cycle Over and reset all bits
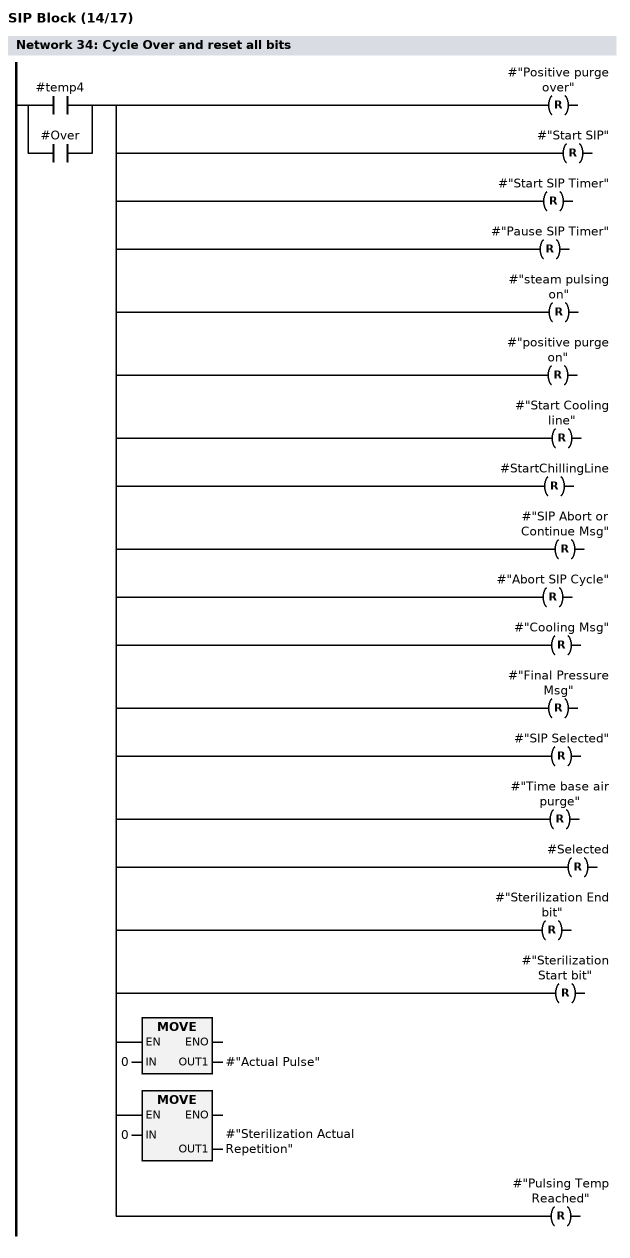
   RUNG wire#powerrail
      Contact( #temp4 )
      wire#w1
      R_Coil( #"Positive purge over" )
   END_RUNG
   RUNG wire#powerrail
      Contact( #Over )
   END_RUNG wire#w1
   RUNG wire#w1
      R_Coil( #"Start SIP" )
   END_RUNG
   RUNG wire#w1
      R_Coil( #"Start SIP Timer" )
   END_RUNG
   RUNG wire#w1
      R_Coil( #"Pause SIP Timer" )
   END_RUNG
   RUNG wire#w1
      R_Coil( #"steam pulsing on" )
   END_RUNG
   RUNG wire#w1
      R_Coil( #"positive purge on" )
   END_RUNG
   RUNG wire#w1
      R_Coil( #"Start Cooling line" )
   END_RUNG
   RUNG wire#w1
      R_Coil( #StartChillingLine )
   END_RUNG
   RUNG wire#w1
      R_Coil( #"SIP Abort or Continue Msg" )
   END_RUNG
   RUNG wire#w1
      R_Coil( #"Abort SIP Cycle" )
   END_RUNG
   RUNG wire#w1
      R_Coil( #"Cooling Msg" )
   END_RUNG
   RUNG wire#w1
      R_Coil( #"Final Pressure Msg" )
   END_RUNG
   RUNG wire#w1
      R_Coil( #"SIP Selected" )
   END_RUNG
   RUNG wire#w1
      R_Coil( #"Time base air purge" )
   END_RUNG
   RUNG wire#w1
      R_Coil( #Selected )
   END_RUNG
   RUNG wire#w1
      R_Coil( #"Sterilization End bit" )
   END_RUNG
   RUNG wire#w1
      R_Coil( #"Sterilization Start bit" )
   END_RUNG
   RUNG wire#w1
      { S7_GenerateENO := "TRUE" } Move(in := 0, out1 => #"Actual Pulse")
   END_RUNG
   RUNG wire#w1
      { S7_GenerateENO := "TRUE" } Move(in := 0, out1 => #"Sterilization Actual Repetition")
   END_RUNG
   RUNG wire#w1
      R_Coil( #"Pulsing Temp Reached" )
   END_RUNG
   // the same network as SCL:
   IF #temp4 OR #Over THEN
       #"Positive purge over" := FALSE;
       #"Start SIP" := FALSE;
       #"Start SIP Timer" := FALSE;
       #"Pause SIP Timer" := FALSE;
       #"steam pulsing on" := FALSE;
       #"positive purge on" := FALSE;
       #"Start Cooling line" := FALSE;
       #StartChillingLine := FALSE;
       #"SIP Abort or Continue Msg" := FALSE;
       #"Abort SIP Cycle" := FALSE;
       #"Cooling Msg" := FALSE;
       #"Final Pressure Msg" := FALSE;
       #"SIP Selected" := FALSE;
       #"Time base air purge" := FALSE;
       #Selected := FALSE;
       #"Sterilization End bit" := FALSE;
       #"Sterilization Start bit" := FALSE;
       #"Actual Pulse" := 0;
       #"Sterilization Actual Repetition" := 0;
       #"Pulsing Temp Reached" := FALSE;
   END_IF;
END_REGION

REGION Network 35: Abort
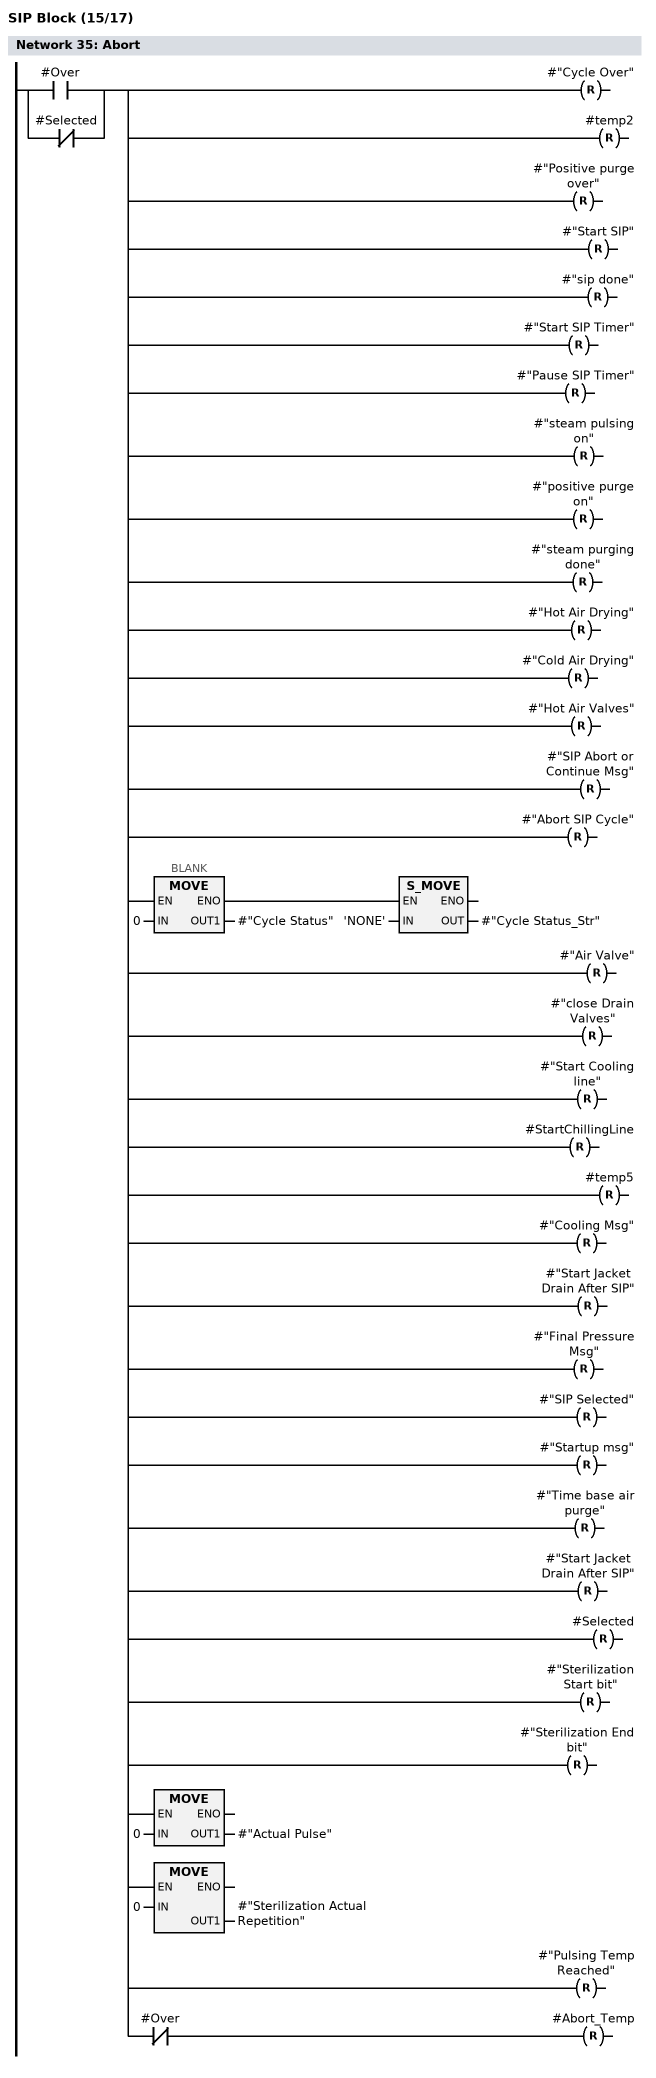
   RUNG wire#powerrail
      Contact( #Over )
      wire#w1
      R_Coil( #"Cycle Over" )
   END_RUNG
   RUNG wire#powerrail
      I_Contact( #Selected )
   END_RUNG wire#w1
   RUNG wire#w1
      R_Coil( #temp2 )
   END_RUNG
   RUNG wire#w1
      R_Coil( #"Positive purge over" )
   END_RUNG
   RUNG wire#w1
      R_Coil( #"Start SIP" )
   END_RUNG
   RUNG wire#w1
      R_Coil( #"sip done" )
   END_RUNG
   RUNG wire#w1
      R_Coil( #"Start SIP Timer" )
   END_RUNG
   RUNG wire#w1
      R_Coil( #"Pause SIP Timer" )
   END_RUNG
   RUNG wire#w1
      R_Coil( #"steam pulsing on" )
   END_RUNG
   RUNG wire#w1
      R_Coil( #"positive purge on" )
   END_RUNG
   RUNG wire#w1
      R_Coil( #"steam purging done" )
   END_RUNG
   RUNG wire#w1
      R_Coil( #"Hot Air Drying" )
   END_RUNG
   RUNG wire#w1
      R_Coil( #"Cold Air Drying" )
   END_RUNG
   RUNG wire#w1
      R_Coil( #"Hot Air Valves" )
   END_RUNG
   RUNG wire#w1
      R_Coil( #"SIP Abort or Continue Msg" )
   END_RUNG
   RUNG wire#w1
      R_Coil( #"Abort SIP Cycle" )
   END_RUNG
   RUNG wire#w1
      { S7_GenerateENO := "TRUE" } Move(in := 0, out1 => #"Cycle Status")   // BLANK
      S_Move(in := 'NONE', out => #"Cycle Status_Str")
   END_RUNG
   RUNG wire#w1
      R_Coil( #"Air Valve" )
   END_RUNG
   RUNG wire#w1
      R_Coil( #"close Drain Valves" )
   END_RUNG
   RUNG wire#w1
      R_Coil( #"Start Cooling line" )
   END_RUNG
   RUNG wire#w1
      R_Coil( #StartChillingLine )
   END_RUNG
   RUNG wire#w1
      R_Coil( #temp5 )
   END_RUNG
   RUNG wire#w1
      R_Coil( #"Cooling Msg" )
   END_RUNG
   RUNG wire#w1
      R_Coil( #"Start Jacket Drain After SIP" )
   END_RUNG
   RUNG wire#w1
      R_Coil( #"Final Pressure Msg" )
   END_RUNG
   RUNG wire#w1
      R_Coil( #"SIP Selected" )
   END_RUNG
   RUNG wire#w1
      R_Coil( #"Startup msg" )
   END_RUNG
   RUNG wire#w1
      R_Coil( #"Time base air purge" )
   END_RUNG
   RUNG wire#w1
      R_Coil( #"Start Jacket Drain After SIP" )
   END_RUNG
   RUNG wire#w1
      R_Coil( #Selected )
   END_RUNG
   RUNG wire#w1
      R_Coil( #"Sterilization Start bit" )
   END_RUNG
   RUNG wire#w1
      R_Coil( #"Sterilization End bit" )
   END_RUNG
   RUNG wire#w1
      { S7_GenerateENO := "TRUE" } Move(in := 0, out1 => #"Actual Pulse")
   END_RUNG
   RUNG wire#w1
      { S7_GenerateENO := "TRUE" } Move(in := 0, out1 => #"Sterilization Actual Repetition")
   END_RUNG
   RUNG wire#w1
      R_Coil( #"Pulsing Temp Reached" )
   END_RUNG
   RUNG wire#w1
      I_Contact( #Over )
      R_Coil( #Abort_Temp )
   END_RUNG
   // the same network as SCL:
   // ENO of a box is taken as its EN; it also drops when the box reports an error
   #_w1 := #Over OR NOT #Selected;
   IF #_w1 THEN
       #"Cycle Over" := FALSE;
       #temp2 := FALSE;
       #"Positive purge over" := FALSE;
       #"Start SIP" := FALSE;
       #"sip done" := FALSE;
       #"Start SIP Timer" := FALSE;
       #"Pause SIP Timer" := FALSE;
       #"steam pulsing on" := FALSE;
       #"positive purge on" := FALSE;
       #"steam purging done" := FALSE;
       #"Hot Air Drying" := FALSE;
       #"Cold Air Drying" := FALSE;
       #"Hot Air Valves" := FALSE;
       #"SIP Abort or Continue Msg" := FALSE;
       #"Abort SIP Cycle" := FALSE;
       #"Cycle Status" := 0;   // BLANK
       #"Cycle Status_Str" := 'NONE';
       #"Air Valve" := FALSE;
       #"close Drain Valves" := FALSE;
       #"Start Cooling line" := FALSE;
       #StartChillingLine := FALSE;
       #temp5 := FALSE;
       #"Cooling Msg" := FALSE;
       #"Start Jacket Drain After SIP" := FALSE;
       #"Final Pressure Msg" := FALSE;
       #"SIP Selected" := FALSE;
       #"Startup msg" := FALSE;
       #"Time base air purge" := FALSE;
       #"Start Jacket Drain After SIP" := FALSE;
       #Selected := FALSE;
       #"Sterilization Start bit" := FALSE;
       #"Sterilization End bit" := FALSE;
       #"Actual Pulse" := 0;
       #"Sterilization Actual Repetition" := 0;
       #"Pulsing Temp Reached" := FALSE;
   END_IF;
   IF #_w1 AND NOT #Over THEN #Abort_Temp := FALSE; END_IF;
END_REGION

REGION Network 36: #"Cip drain valves" during steam purging
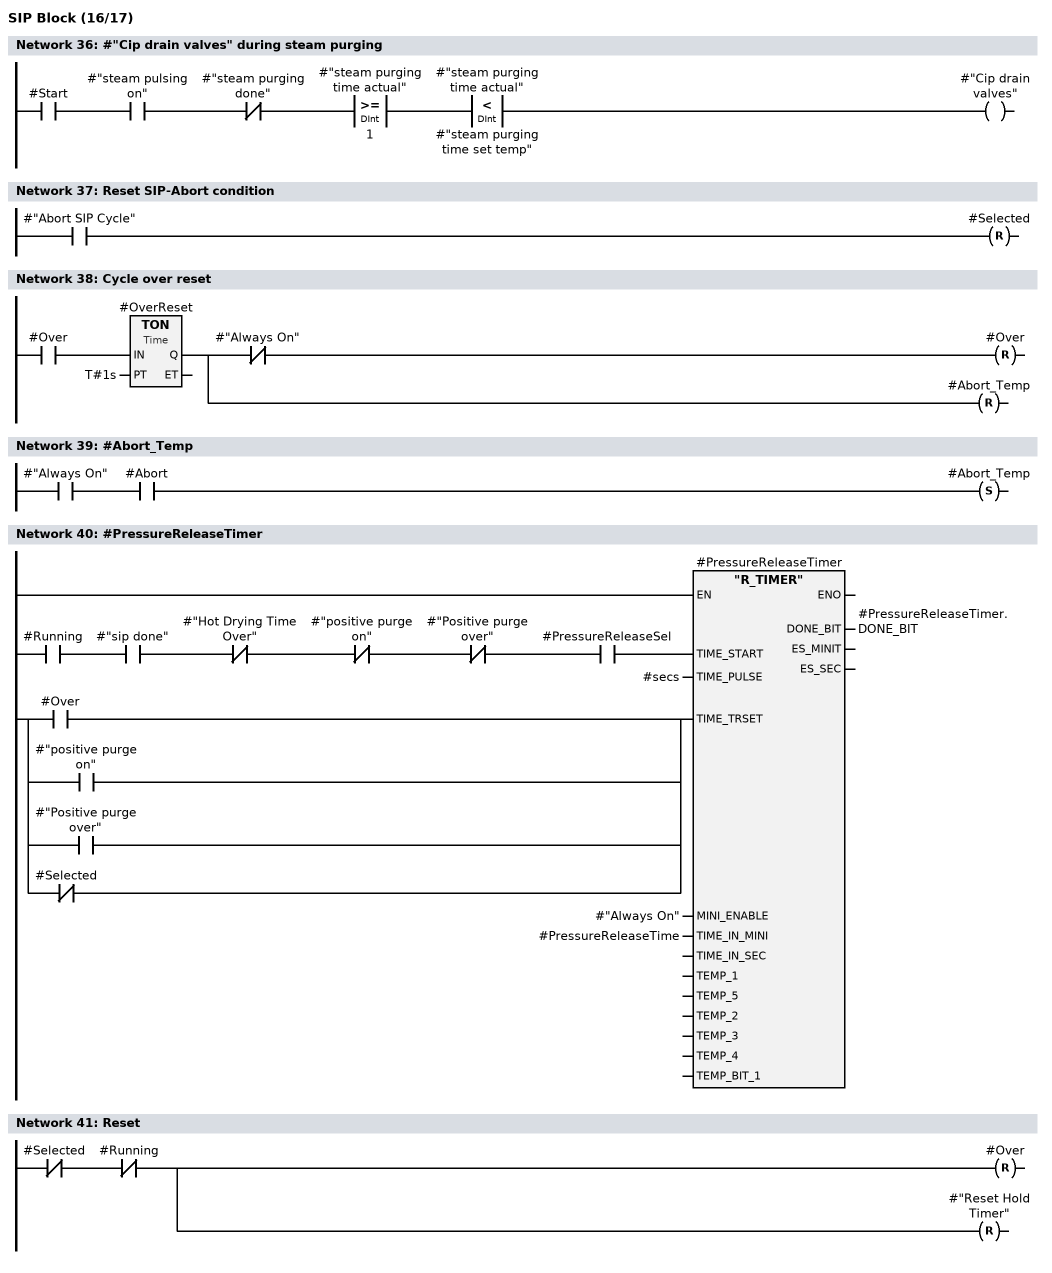
   RUNG wire#powerrail
      Contact( #Start )
      Contact( #"steam pulsing on" )
      I_Contact( #"steam purging done" )
      { S7_Templates := "SrcType := DInt" } GE_Contact(in1 := #"steam purging time actual", in2 := 1)
      { S7_Templates := "SrcType := DInt" } LT_Contact(in1 := #"steam purging time actual", in2 := #"steam purging time set temp")
      Coil( #"Cip drain valves" )
   END_RUNG
   // the same network as SCL:
   #"Cip drain valves" := #Start AND #"steam pulsing on" AND NOT #"steam purging done" AND (#"steam purging time actual" >= 1) AND (#"steam purging time actual" < #"steam purging time set temp");
END_REGION

REGION Network 37: Reset SIP-Abort condition
   RUNG wire#powerrail
      Contact( #"Abort SIP Cycle" )
      R_Coil( #Selected )
   END_RUNG
   // the same network as SCL:
   IF #"Abort SIP Cycle" THEN #Selected := FALSE; END_IF;
END_REGION

REGION Network 38: Cycle over reset
   RUNG wire#powerrail
      Contact( #Over )
      { S7_Templates := "time_type := Time" } #OverReset.TON(pt := T#1s, et =>)
      wire#w1
      I_Contact( #"Always On" )
      R_Coil( #Over )
   END_RUNG
   RUNG wire#w1
      R_Coil( #Abort_Temp )
   END_RUNG
   // the same network as SCL:
   #OverReset.TON(IN := #Over, PT := T#1s);
   IF #OverReset.Q AND NOT #"Always On" THEN #Over := FALSE; END_IF;
   IF #OverReset.Q THEN #Abort_Temp := FALSE; END_IF;
END_REGION

REGION Network 39: #Abort_Temp
   RUNG wire#powerrail
      Contact( #"Always On" )
      Contact( #Abort )
      S_Coil( #Abort_Temp )
   END_RUNG
   // the same network as SCL:
   IF #"Always On" AND #Abort THEN #Abort_Temp := TRUE; END_IF;
END_REGION

REGION Network 40: #PressureReleaseTimer
   RUNG wire#powerrail
      #PressureReleaseTimer(TIME_START := wire#w1, TIME_TRSET := wire#w2, TIME_PULSE := #secs, MINI_ENABLE := #"Always On", TIME_IN_MINI := #PressureReleaseTime, TIME_IN_SEC :=, TEMP_1 :=, TEMP_5 :=, TEMP_2 :=, TEMP_3 :=, TEMP_4 :=, TEMP_BIT_1 :=, DONE_BIT => #PressureReleaseTimer.DONE_BIT, ES_MINIT =>, ES_SEC =>)
   END_RUNG
   RUNG wire#powerrail
      Contact( #Running )
      Contact( #"sip done" )
      I_Contact( #"Hot Drying Time Over" )
      I_Contact( #"positive purge on" )
      I_Contact( #"Positive purge over" )
      Contact( #PressureReleaseSel )
   END_RUNG wire#w1
   RUNG wire#powerrail
      Contact( #Over )
   END_RUNG wire#w2
   RUNG wire#powerrail
      Contact( #"positive purge on" )
   END_RUNG wire#w2
   RUNG wire#powerrail
      Contact( #"Positive purge over" )
   END_RUNG wire#w2
   RUNG wire#powerrail
      I_Contact( #Selected )
   END_RUNG wire#w2
   // the same network as SCL:
   #PressureReleaseTimer(TIME_START := #Running AND #"sip done" AND NOT #"Hot Drying Time Over" AND NOT #"positive purge on" AND NOT #"Positive purge over" AND #PressureReleaseSel,   // "R_TIMER"
                         TIME_PULSE := #secs,
                         TIME_TRSET := #Over OR #"positive purge on" OR #"Positive purge over" OR NOT #Selected,
                         MINI_ENABLE := #"Always On",
                         TIME_IN_MINI := #PressureReleaseTime,
                         DONE_BIT => #PressureReleaseTimer.DONE_BIT);
END_REGION

REGION Network 41: Reset
   RUNG wire#powerrail
      I_Contact( #Selected )
      I_Contact( #Running )
      wire#w1
      R_Coil( #Over )
   END_RUNG
   RUNG wire#w1
      R_Coil( #"Reset Hold Timer" )
   END_RUNG
   // the same network as SCL:
   IF NOT #Selected AND NOT #Running THEN
       #Over := FALSE;
       #"Reset Hold Timer" := FALSE;
   END_IF;
END_REGION

REGION Network 42: #"Sterilization Set RepetitionTemp"
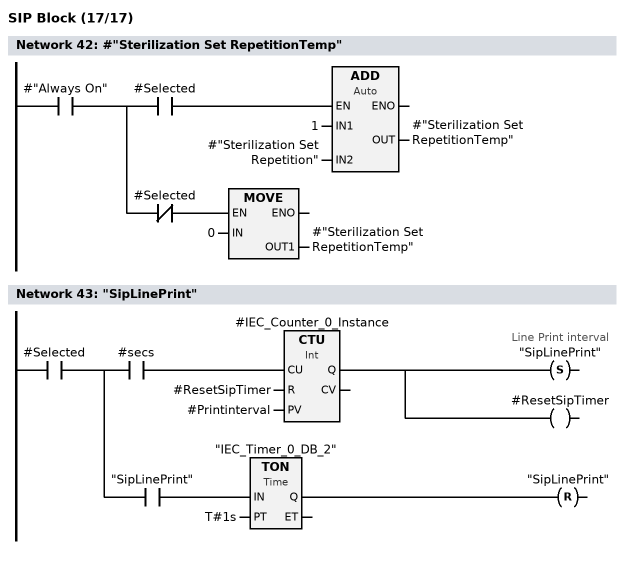
   RUNG wire#powerrail
      Contact( #"Always On" )
      wire#w1
      Contact( #Selected )
      Add(in1 := 1, in2 := #"Sterilization Set Repetition", out => #"Sterilization Set RepetitionTemp")
   END_RUNG
   RUNG wire#w1
      I_Contact( #Selected )
      Move(in := 0, out1 => #"Sterilization Set RepetitionTemp")
   END_RUNG
   // the same network as SCL:
   IF #"Always On" AND #Selected THEN
       #"Sterilization Set RepetitionTemp" := 1 + #"Sterilization Set Repetition";
   END_IF;
   IF #"Always On" AND NOT #Selected THEN #"Sterilization Set RepetitionTemp" := 0; END_IF;
END_REGION

REGION Network 43: "SipLinePrint"
   RUNG wire#powerrail
      Contact( #Selected )
      wire#w1
      Contact( #secs )
      { S7_Templates := "value_type := Int" } #IEC_Counter_0_Instance.CTU(r := #ResetSipTimer, pv := #Printinterval, cv =>)
      wire#w2
      S_Coil( "SipLinePrint" )   // Line Print interval
   END_RUNG
   RUNG wire#w2
      Coil( #ResetSipTimer )
   END_RUNG
   RUNG wire#w1
      Contact( "SipLinePrint" )
      { S7_Templates := "time_type := Time" } "IEC_Timer_0_DB_2".TON(pt := T#1s, et =>)
      R_Coil( "SipLinePrint" )
   END_RUNG
   // the same network as SCL:
   #IEC_Counter_0_Instance(CU := #Selected AND #secs, R := #ResetSipTimer, PV := #Printinterval);   // CTU
   IF #IEC_Counter_0_Instance.Q THEN
       "SipLinePrint" := TRUE;   // Line Print interval
   END_IF;
   #ResetSipTimer := #IEC_Counter_0_Instance.Q;
   "IEC_Timer_0_DB_2".TON(IN := #Selected AND "SipLinePrint", PT := T#1s);
   IF "IEC_Timer_0_DB_2".Q THEN "SipLinePrint" := FALSE; END_IF;
END_REGION
END_FUNCTION_BLOCK

FUNCTION_BLOCK "SIP TEMPERATURE CONTROLER"   // FB502, LAD
{ S7_Optimized_Access := 'FALSE' }
// stored: AutoNumber false, SetENOAutomatically false
   VAR_INPUT
      "CONROL ON" : Bool;
      Second_Pulse : Bool;
      Actual_sip_temp : Real;
      "SET  TEMPERATUR" : Real;
      "TEMPERATURE RANGE_1" : Real;
      "TEMPERATURE RANGE_2" : Real;
      "TEMPERATURE RANGE_4" : Real;
      "TEMPERATURE RANGE_6" : Real;
      "TEMPERATURE RANGE_8" : Real;
      ON_SEC_1 { ExternalAccessible := 'False'; ExternalVisible := 'False'; ExternalWritable := 'False'} : Int;
      ON_SEC_2 { ExternalAccessible := 'False'; ExternalVisible := 'False'; ExternalWritable := 'False'} : Int;
      ON_SEC_3 { ExternalAccessible := 'False'; ExternalVisible := 'False'; ExternalWritable := 'False'} : Int;
      ON_SEC_4 { ExternalAccessible := 'False'; ExternalVisible := 'False'; ExternalWritable := 'False'} : Int;
      OFF_SEC_1 { ExternalAccessible := 'False'; ExternalVisible := 'False'; ExternalWritable := 'False'} : Int;
      OFF_SEC_2 { ExternalAccessible := 'False'; ExternalVisible := 'False'; ExternalWritable := 'False'} : Int;
      OFF_SEC_3 { ExternalAccessible := 'False'; ExternalVisible := 'False'; ExternalWritable := 'False'} : Int;
      OFF_SEC_4 { ExternalAccessible := 'False'; ExternalVisible := 'False'; ExternalWritable := 'False'} : Int;
      RESET_BIT : Bool;
   END_VAR
   VAR_OUTPUT
      "VALVE CONTROL" : Bool;
      TEMPPERATUR_REACHED : Bool;
   END_VAR
   VAR_IN_OUT
      ON_SEC : Int;
      OFF_SEC : Int;
      ON_SEC_TIME : Int;
      OFF_SEC_TIME : Int;
      TEMP_1 : Bool;
   END_VAR
   VAR_TEMP   // added for the SCL form of the ladder/FBD networks
      _w1 : Bool;
      _w2 : Bool;
      _w3 : Bool;
   END_VAR
BEGIN

REGION Network 1: range
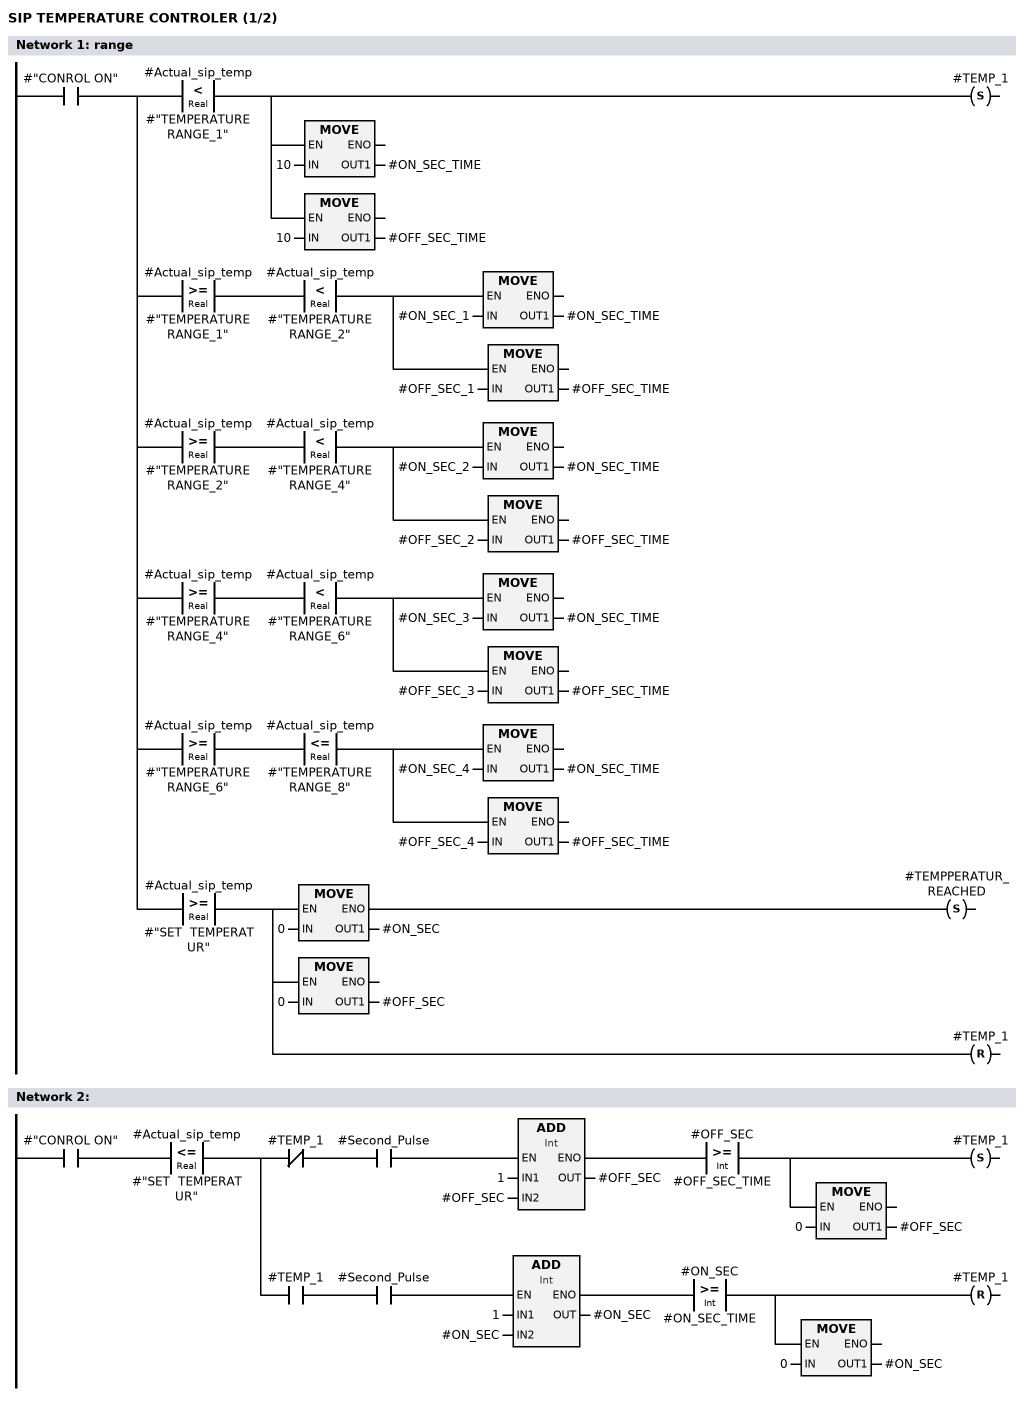
   RUNG wire#powerrail
      Contact( #"CONROL ON" )
      wire#w1
      { S7_Templates := "SrcType := Real" } LT_Contact(in1 := #Actual_sip_temp, in2 := #"TEMPERATURE RANGE_1")
      wire#w2
      S_Coil( #TEMP_1 )
   END_RUNG
   RUNG wire#w2
      { S7_GenerateENO := "TRUE" } Move(in := 10, out1 => #ON_SEC_TIME)
   END_RUNG
   RUNG wire#w2
      { S7_GenerateENO := "TRUE" } Move(in := 10, out1 => #OFF_SEC_TIME)
   END_RUNG
   RUNG wire#w1
      { S7_Templates := "SrcType := Real" } GE_Contact(in1 := #Actual_sip_temp, in2 := #"TEMPERATURE RANGE_1")
      { S7_Templates := "SrcType := Real" } LT_Contact(in1 := #Actual_sip_temp, in2 := #"TEMPERATURE RANGE_2")
      wire#w3
      { S7_GenerateENO := "TRUE" } Move(in := #ON_SEC_1, out1 => #ON_SEC_TIME)
   END_RUNG
   RUNG wire#w3
      { S7_GenerateENO := "TRUE" } Move(in := #OFF_SEC_1, out1 => #OFF_SEC_TIME)
   END_RUNG
   RUNG wire#w1
      { S7_Templates := "SrcType := Real" } GE_Contact(in1 := #Actual_sip_temp, in2 := #"TEMPERATURE RANGE_2")
      { S7_Templates := "SrcType := Real" } LT_Contact(in1 := #Actual_sip_temp, in2 := #"TEMPERATURE RANGE_4")
      wire#w4
      { S7_GenerateENO := "TRUE" } Move(in := #ON_SEC_2, out1 => #ON_SEC_TIME)
   END_RUNG
   RUNG wire#w4
      { S7_GenerateENO := "TRUE" } Move(in := #OFF_SEC_2, out1 => #OFF_SEC_TIME)
   END_RUNG
   RUNG wire#w1
      { S7_Templates := "SrcType := Real" } GE_Contact(in1 := #Actual_sip_temp, in2 := #"TEMPERATURE RANGE_4")
      { S7_Templates := "SrcType := Real" } LT_Contact(in1 := #Actual_sip_temp, in2 := #"TEMPERATURE RANGE_6")
      wire#w5
      { S7_GenerateENO := "TRUE" } Move(in := #ON_SEC_3, out1 => #ON_SEC_TIME)
   END_RUNG
   RUNG wire#w5
      { S7_GenerateENO := "TRUE" } Move(in := #OFF_SEC_3, out1 => #OFF_SEC_TIME)
   END_RUNG
   RUNG wire#w1
      { S7_Templates := "SrcType := Real" } GE_Contact(in1 := #Actual_sip_temp, in2 := #"TEMPERATURE RANGE_6")
      { S7_Templates := "SrcType := Real" } LE_Contact(in1 := #Actual_sip_temp, in2 := #"TEMPERATURE RANGE_8")
      wire#w6
      { S7_GenerateENO := "TRUE" } Move(in := #ON_SEC_4, out1 => #ON_SEC_TIME)
   END_RUNG
   RUNG wire#w6
      { S7_GenerateENO := "TRUE" } Move(in := #OFF_SEC_4, out1 => #OFF_SEC_TIME)
   END_RUNG
   RUNG wire#w1
      { S7_Templates := "SrcType := Real" } GE_Contact(in1 := #Actual_sip_temp, in2 := #"SET  TEMPERATUR")
      wire#w7
      { S7_GenerateENO := "TRUE" } Move(in := 0, out1 => #ON_SEC)
      S_Coil( #TEMPPERATUR_REACHED )
   END_RUNG
   RUNG wire#w7
      { S7_GenerateENO := "TRUE" } Move(in := 0, out1 => #OFF_SEC)
   END_RUNG
   RUNG wire#w7
      R_Coil( #TEMP_1 )
   END_RUNG
   // the same network as SCL:
   // ENO of a box is taken as its EN; it also drops when the box reports an error
   IF #"CONROL ON" AND (#Actual_sip_temp < #"TEMPERATURE RANGE_1") THEN
       #TEMP_1 := TRUE;
       #ON_SEC_TIME := 10;
       #OFF_SEC_TIME := 10;
   END_IF;
   IF #"CONROL ON" AND (#Actual_sip_temp >= #"TEMPERATURE RANGE_1") AND (#Actual_sip_temp < #"TEMPERATURE RANGE_2") THEN
       #ON_SEC_TIME := #ON_SEC_1;
       #OFF_SEC_TIME := #OFF_SEC_1;
   END_IF;
   IF #"CONROL ON" AND (#Actual_sip_temp >= #"TEMPERATURE RANGE_2") AND (#Actual_sip_temp < #"TEMPERATURE RANGE_4") THEN
       #ON_SEC_TIME := #ON_SEC_2;
       #OFF_SEC_TIME := #OFF_SEC_2;
   END_IF;
   IF #"CONROL ON" AND (#Actual_sip_temp >= #"TEMPERATURE RANGE_4") AND (#Actual_sip_temp < #"TEMPERATURE RANGE_6") THEN
       #ON_SEC_TIME := #ON_SEC_3;
       #OFF_SEC_TIME := #OFF_SEC_3;
   END_IF;
   IF #"CONROL ON" AND (#Actual_sip_temp >= #"TEMPERATURE RANGE_6") AND (#Actual_sip_temp <= #"TEMPERATURE RANGE_8") THEN
       #ON_SEC_TIME := #ON_SEC_4;
       #OFF_SEC_TIME := #OFF_SEC_4;
   END_IF;
   IF #"CONROL ON" AND (#Actual_sip_temp >= #"SET  TEMPERATUR") THEN
       #ON_SEC := 0;
       #TEMPPERATUR_REACHED := TRUE;
       #OFF_SEC := 0;
       #TEMP_1 := FALSE;
   END_IF;
END_REGION

REGION Network 2
   RUNG wire#powerrail
      Contact( #"CONROL ON" )
      { S7_Templates := "SrcType := Real" } LE_Contact(in1 := #Actual_sip_temp, in2 := #"SET  TEMPERATUR")
      wire#w1
      I_Contact( #TEMP_1 )
      Contact( #Second_Pulse )
      { S7_Templates := "SrcType := Int"; S7_GenerateENO := "TRUE" } Add(in1 := 1, in2 := #OFF_SEC, out => #OFF_SEC)
      { S7_Templates := "SrcType := Int" } GE_Contact(in1 := #OFF_SEC, in2 := #OFF_SEC_TIME)
      wire#w2
      S_Coil( #TEMP_1 )
   END_RUNG
   RUNG wire#w2
      { S7_GenerateENO := "TRUE" } Move(in := 0, out1 => #OFF_SEC)
   END_RUNG
   RUNG wire#w1
      Contact( #TEMP_1 )
      Contact( #Second_Pulse )
      { S7_Templates := "SrcType := Int"; S7_GenerateENO := "TRUE" } Add(in1 := 1, in2 := #ON_SEC, out => #ON_SEC)
      { S7_Templates := "SrcType := Int" } GE_Contact(in1 := #ON_SEC, in2 := #ON_SEC_TIME)
      wire#w3
      R_Coil( #TEMP_1 )
   END_RUNG
   RUNG wire#w3
      { S7_GenerateENO := "TRUE" } Move(in := 0, out1 => #ON_SEC)
   END_RUNG
   // the same network as SCL:
   // ENO of a box is taken as its EN; it also drops when the box reports an error
   #_w1 := #"CONROL ON" AND (#Actual_sip_temp <= #"SET  TEMPERATUR");
   #_w2 := #_w1 AND NOT #TEMP_1 AND #Second_Pulse;
   IF #_w2 THEN #OFF_SEC := 1 + #OFF_SEC; END_IF;
   IF #_w2 AND (#OFF_SEC >= #OFF_SEC_TIME) THEN
       #TEMP_1 := TRUE;
       #OFF_SEC := 0;
   END_IF;
   #_w3 := #_w1 AND #TEMP_1 AND #Second_Pulse;
   IF #_w3 THEN #ON_SEC := 1 + #ON_SEC; END_IF;
   IF #_w3 AND (#ON_SEC >= #ON_SEC_TIME) THEN
       #TEMP_1 := FALSE;
       #ON_SEC := 0;
   END_IF;
END_REGION

REGION Network 3
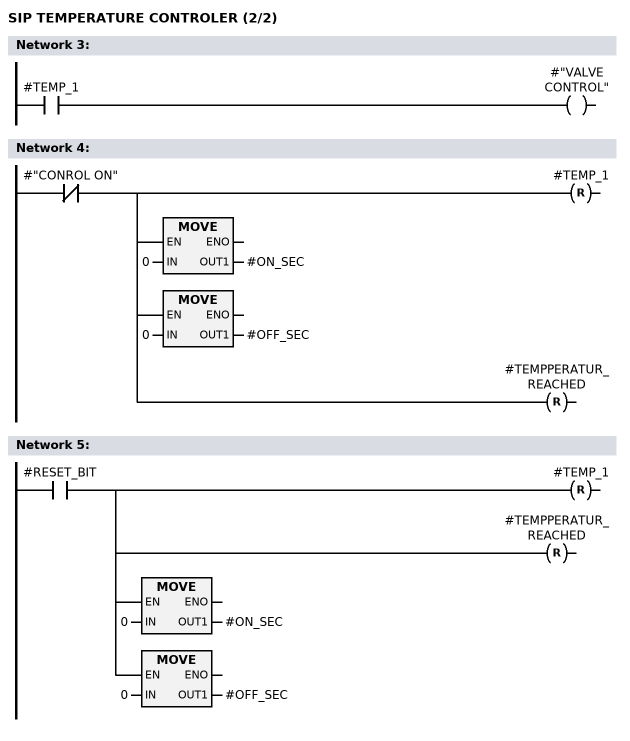
   RUNG wire#powerrail
      Contact( #TEMP_1 )
      Coil( #"VALVE CONTROL" )
   END_RUNG
   // the same network as SCL:
   #"VALVE CONTROL" := #TEMP_1;
END_REGION

REGION Network 4
   RUNG wire#powerrail
      I_Contact( #"CONROL ON" )
      wire#w1
      R_Coil( #TEMP_1 )
   END_RUNG
   RUNG wire#w1
      { S7_GenerateENO := "TRUE" } Move(in := 0, out1 => #ON_SEC)
   END_RUNG
   RUNG wire#w1
      { S7_GenerateENO := "TRUE" } Move(in := 0, out1 => #OFF_SEC)
   END_RUNG
   RUNG wire#w1
      R_Coil( #TEMPPERATUR_REACHED )
   END_RUNG
   // the same network as SCL:
   IF NOT #"CONROL ON" THEN
       #TEMP_1 := FALSE;
       #ON_SEC := 0;
       #OFF_SEC := 0;
       #TEMPPERATUR_REACHED := FALSE;
   END_IF;
END_REGION

REGION Network 5
   RUNG wire#powerrail
      Contact( #RESET_BIT )
      wire#w1
      R_Coil( #TEMP_1 )
   END_RUNG
   RUNG wire#w1
      R_Coil( #TEMPPERATUR_REACHED )
   END_RUNG
   RUNG wire#w1
      { S7_GenerateENO := "TRUE" } Move(in := 0, out1 => #ON_SEC)
   END_RUNG
   RUNG wire#w1
      { S7_GenerateENO := "TRUE" } Move(in := 0, out1 => #OFF_SEC)
   END_RUNG
   // the same network as SCL:
   IF #RESET_BIT THEN
       #TEMP_1 := FALSE;
       #TEMPPERATUR_REACHED := FALSE;
       #ON_SEC := 0;
       #OFF_SEC := 0;
   END_IF;
END_REGION
END_FUNCTION_BLOCK

FUNCTION_BLOCK "VesselLamp"   // FB7, LAD
{ S7_Optimized_Access := 'FALSE' }
// stored: AutoNumber false, SetENOAutomatically false
   VAR_INPUT
      Secs : Bool;
      AlwaysTrue : Bool;
      AlwaysFalse : Bool;
   END_VAR
   VAR_OUTPUT
      DONE_BIT : Bool;
      ES_MINIT : DInt;
      ES_SEC : DInt;
   END_VAR
   VAR
      LF01 { S7_SetPoint := 'True'} : "TIMER";   // LF01
   END_VAR
BEGIN

REGION Network 1: #VslLamp01
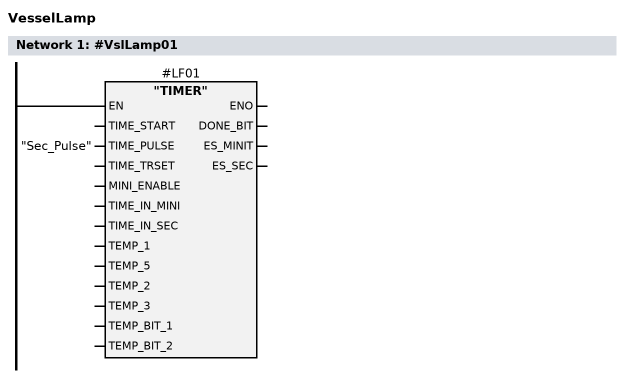
   RUNG wire#powerrail
      #LF01(TIME_START :=, TIME_PULSE := "Sec_Pulse", TIME_TRSET :=, MINI_ENABLE :=, TIME_IN_MINI :=, TIME_IN_SEC :=, TEMP_1 :=, TEMP_5 :=, TEMP_2 :=, TEMP_3 :=, TEMP_BIT_1 :=, TEMP_BIT_2 :=, DONE_BIT =>, ES_MINIT =>, ES_SEC =>)
   END_RUNG
   // the same network as SCL:
   #LF01(TIME_PULSE := "Sec_Pulse");   // "TIMER"
END_REGION
END_FUNCTION_BLOCK

FUNCTION "Loadcell_Profinet" : Void   // FC37, LAD
{ S7_Optimized_Access := 'TRUE' }
// stored: SetENOAutomatically false
BEGIN

REGION Network 1: LoadcellCV15
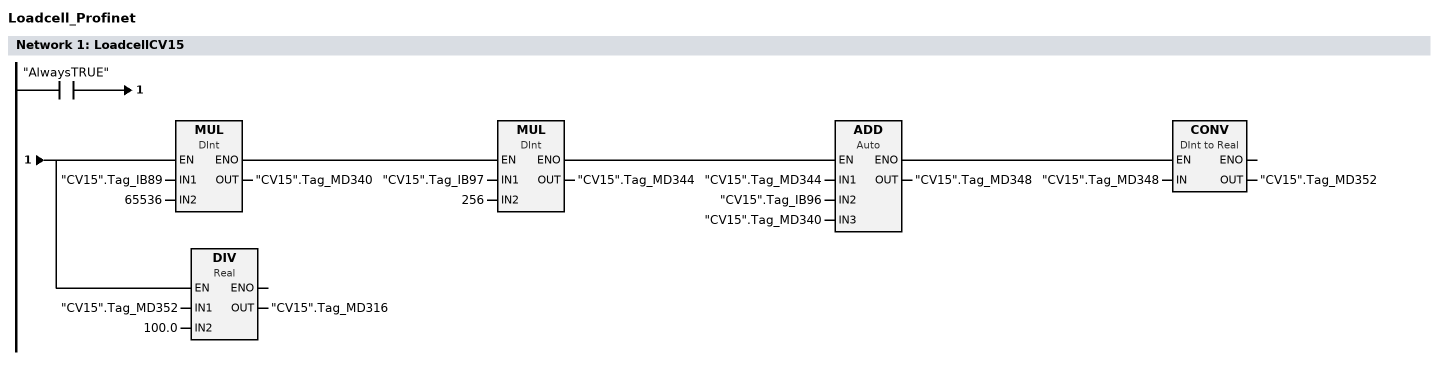
   RUNG wire#powerrail
      Contact( "AlwaysTRUE" )
      wire#w1
      { S7_Templates := "SrcType := DInt" } Mul(in1 := "CV15".Tag_IB89, in2 := 65536, out => "CV15".Tag_MD340)
      { S7_Templates := "SrcType := DInt" } Mul(in1 := "CV15".Tag_IB97, in2 := 256, out => "CV15".Tag_MD344)
      Add(in1 := "CV15".Tag_MD344, in2 := "CV15".Tag_IB96, in3 := "CV15".Tag_MD340, out => "CV15".Tag_MD348)
      { S7_Templates := "[SrcType := DInt, DestType := Real]" } Convert(in := "CV15".Tag_MD348, out => "CV15".Tag_MD352)
   END_RUNG
   RUNG wire#w1
      { S7_Templates := "SrcType := Real" } Div(in1 := "CV15".Tag_MD352, in2 := 100.0, out => "CV15".Tag_MD316)
   END_RUNG
   // the same network as SCL:
   IF "AlwaysTRUE" THEN
       "CV15".Tag_MD340 := "CV15".Tag_IB89 * 65536;
       "CV15".Tag_MD344 := "CV15".Tag_IB97 * 256;
       "CV15".Tag_MD348 := "CV15".Tag_MD344 + "CV15".Tag_IB96 + "CV15".Tag_MD340;
       "CV15".Tag_MD352 := DINT_TO_REAL("CV15".Tag_MD348);
       "CV15".Tag_MD316 := "CV15".Tag_MD352 / 100.0;
   END_IF;
END_REGION
END_FUNCTION

DATA_BLOCK "BatchDetailsLength_DB"   // DB40
// stored: InstanceOfName BatchDetailsLength, InstanceOfType FB
"BatchDetailsLength"
BEGIN
END_DATA_BLOCK

DATA_BLOCK "BATCH LINE PRINT_DB"   // DB14
// stored: InstanceOfName BATCH LINE PRINT, InstanceOfType FB
"BATCH LINE PRINT"
BEGIN
END_DATA_BLOCK

DATA_BLOCK "BatchTempOnOff"   // DB300
// stored: AutoNumber false, InstanceOfName FB104, InstanceOfType FB
"FB104"
BEGIN
END_DATA_BLOCK

DATA_BLOCK "FillWfi"   // DB302
AUTHOR : PRECISE
FAMILY : PRECISE
// stored: AutoNumber false, InstanceOfName FB301, InstanceOfType FB
"FB301"
BEGIN
END_DATA_BLOCK

DATA_BLOCK "FinalVolumeMakeup"   // DB313
AUTHOR : PRECISE
FAMILY : PRECISE
// stored: AutoNumber false, InstanceOfName FB301, InstanceOfType FB
"FB301"
BEGIN
END_DATA_BLOCK

DATA_BLOCK "GasBlanketing"   // DB308
AUTHOR : PRECISE
FAMILY : PRECISE
// stored: AutoNumber false, InstanceOfName FB304, InstanceOfType FB
"FB304"
BEGIN
END_DATA_BLOCK

DATA_BLOCK "JacketDrain"   // DB312
AUTHOR : PRECISE
FAMILY : PRECISE
// stored: AutoNumber false, InstanceOfName FB317, InstanceOfType FB
"FB317"
BEGIN
END_DATA_BLOCK

DATA_BLOCK "JacketVent"   // DB311
AUTHOR : PRECISE
FAMILY : PRECISE
// stored: AutoNumber false, InstanceOfName FB318, InstanceOfType FB
"FB318"
BEGIN
END_DATA_BLOCK

DATA_BLOCK "Mm01Mixing"   // DB306
AUTHOR : PRECISE
FAMILY : PRECISE
// stored: AutoNumber false, InstanceOfName FB302, InstanceOfType FB
"FB302"
BEGIN
END_DATA_BLOCK

DATA_BLOCK "N2Sparging"   // DB307
AUTHOR : PRECISE
FAMILY : PRECISE
// stored: AutoNumber false, InstanceOfName FB303, InstanceOfType FB
"FB303"
BEGIN
END_DATA_BLOCK

DATA_BLOCK "ProductRecicrulation"   // DB316
AUTHOR : PRECISE
FAMILY : PRECISE
// stored: AutoNumber false, InstanceOfName FB302, InstanceOfType FB
"FB302"
BEGIN
END_DATA_BLOCK

DATA_BLOCK "ProductTransfer"   // DB310
// stored: AutoNumber false, InstanceOfName FB305, InstanceOfType FB
"FB305"
BEGIN
END_DATA_BLOCK

DATA_BLOCK "RMAdd"   // DB305
AUTHOR : PRECISE
FAMILY : PRECISE
// stored: AutoNumber false, InstanceOfName FB310, InstanceOfType FB
"FB310"
BEGIN
END_DATA_BLOCK

DATA_BLOCK "TemperatureControl"   // DB303
AUTHOR : PRECISE
FAMILY : PRECISE
// stored: AutoNumber false, InstanceOfName FB311, InstanceOfType FB
"FB311"
BEGIN
END_DATA_BLOCK

DATA_BLOCK "TemperatureControlValve"   // DB304
// stored: AutoNumber false, InstanceOfName FB104, InstanceOfType FB
"FB104"
BEGIN
END_DATA_BLOCK

DATA_BLOCK "CP01"   // DB23
// stored: InstanceOfName FB614, InstanceOfType FB
"FB614"
BEGIN
END_DATA_BLOCK

DATA_BLOCK "MV3000LineAnimationDb"   // DB801
// stored: AutoNumber false, InstanceOfName MV3000LineAnimation, InstanceOfType FB
"MV3000LineAnimation"
BEGIN
END_DATA_BLOCK

DATA_BLOCK "Pht_Block"   // DB1230
// stored: InstanceOfName PHT Block, InstanceOfType FB
"PHT Block"
BEGIN
END_DATA_BLOCK

DATA_BLOCK "DB603"   // DB603
TITLE = DB603
AUTHOR : PRECISE
FAMILY : PRECISE
// CycleSelection
// stored: AutoNumber false, InstanceOfName FB603, InstanceOfType FB
"FB603"
BEGIN
END_DATA_BLOCK

DATA_BLOCK "DB604"   // DB604
TITLE = DB604
AUTHOR : PRECISE
FAMILY : PRECISE
// CIP FILLING
// stored: AutoNumber false, InstanceOfName FB604, InstanceOfType FB
"FB604"
BEGIN
END_DATA_BLOCK

DATA_BLOCK "DB607"   // DB607
AUTHOR : PRECISE
FAMILY : PRECISE
// stored: AutoNumber false, InstanceOfName FB607, InstanceOfType FB
"FB607"
BEGIN
END_DATA_BLOCK

DATA_BLOCK "DB608"   // DB608
TITLE = DB608
AUTHOR : PRECISE
FAMILY : PRECISE
// CIP RECIRCULATION
// stored: AutoNumber false, InstanceOfName FB608, InstanceOfType FB
"FB608"
BEGIN
END_DATA_BLOCK

DATA_BLOCK "DB609"   // DB609
AUTHOR : PRECISE
FAMILY : PRECISE
// stored: AutoNumber false, InstanceOfName FB609, InstanceOfType FB
"FB609"
BEGIN
END_DATA_BLOCK

DATA_BLOCK "DB610"   // DB610
TITLE = DB610
AUTHOR : PRECISE
FAMILY : PRECISE
// CIP SYSTEM DRAIN
// stored: AutoNumber false, InstanceOfName FB610, InstanceOfType FB
"FB610"
BEGIN
END_DATA_BLOCK

DATA_BLOCK "DB611"   // DB611
TITLE = DB611
AUTHOR : PRECISE
FAMILY : PRECISE
// CIP AIR PURGING
// stored: AutoNumber false, InstanceOfName FB611, InstanceOfType FB
"FB611"
BEGIN
   ParaIn.Selections.PressureMode := 1;
END_DATA_BLOCK

DATA_BLOCK "AiDb"   // DB108
// stored: AutoNumber false, InstanceOfName AiFb, InstanceOfType FB
"AiFb"
BEGIN
   Ai01.AlmHighLimit := 150.0;
   Ai01.AlmLowlimit := -15.0;
   Ai01.HighRange := 150.0;
   Ai01.LowRange := -15.0;
   Ai02.AlmHighLimit := 150.0;
   Ai02.AlmLowlimit := -15.0;
   Ai02.HighRange := 150.0;
   Ai02.LowRange := -15.0;
   Ai02.LowAlarmStatus := 0;
   Ai03.AlmHighLimit := 150.0;
   Ai03.AlmLowlimit := -15.0;
   Ai03.HighRange := 150.0;
   Ai03.LowRange := -15.0;
   Ai04.AlmHighLimit := 150.0;
   Ai04.AlmLowlimit := -15.0;
   Ai04.HighRange := 150.0;
   Ai04.LowRange := -15.0;
   Ai04.LowAlarmStatus := 0;
   Ai05.AlmHighLimit := 150.0;
   Ai05.AlmLowlimit := -15.0;
   Ai05.HighRange := 150.0;
   Ai05.LowRange := -15.0;
   Ai05.LowAlarmStatus := 0;
   Ai06.AlmHighLimit := 150.0;
   Ai06.AlmLowlimit := -15.0;
   Ai06.HighRange := 150.0;
   Ai06.LowRange := -15.0;
   Ai06.LowAlarmStatus := 0;
   Ai07.AlmHighLimit := 150.0;
   Ai07.AlmLowlimit := -15.0;
   Ai07.HighRange := 150.0;
   Ai07.LowRange := -15.0;
   Ai08.AlmHighLimit := 150.0;
   Ai08.AlmLowlimit := -15.0;
   Ai08.HighRange := 150.0;
   Ai08.LowRange := -15.0;
   Ai09.AlmHighLimit := 150.0;
   Ai09.AlmLowlimit := -15.0;
   Ai09.HighRange := 150.0;
   Ai09.LowRange := -15.0;
   Ai10.AlmHighLimit := 150.0;
   Ai10.AlmLowlimit := -15.0;
   Ai10.HighRange := 150.0;
   Ai10.LowRange := -15.0;
   Ai11.AlmHighLimit := 5.0;
   Ai11.AlmLowlimit := -1.0;
   Ai11.HighRange := 5.0;
   Ai11.LowRange := -1.0;
   Ai12.AlmHighLimit := 5.0;
   Ai12.AlmLowlimit := -1.0;
   Ai12.HighRange := 5.0;
   Ai12.LowRange := -1.0;
   Ai13.AlmHighLimit := 5.0;
   Ai13.AlmLowlimit := -1.0;
   Ai13.HighRange := 5.0;
   Ai13.LowRange := -1.0;
   Ai14.HighRange := 5.0;
   Ai14.LowRange := -1.0;
   Ai15.HighRange := 100.0;
   Ai15.LowRange := 0.0;
END_DATA_BLOCK

DATA_BLOCK "AoDb"   // DB106
// stored: AutoNumber false, InstanceOfName AoFb, InstanceOfType FB
"AoFb"
BEGIN
   Ao01.MinOperatingRpm := 50.0;
   Ao01.MaxOperatingRpm := 400.0;
   Ao01.MaxRpm := 400.0;
   Ao02.MinOperatingRpm := 800.0;
   Ao02.MaxOperatingRpm := 2880.0;
   Ao02.MaxRpm := 2880.0;
   Ao03.MaxOperatingRpm := 100.0;
   Ao03.MaxRpm := 100.0;
END_DATA_BLOCK

DATA_BLOCK "DigitalOutput_DB"   // DB5
// stored: InstanceOfName DigitalOutput, InstanceOfType FB
"DigitalOutput"
BEGIN
END_DATA_BLOCK

DATA_BLOCK "DigitalOutput_DB_1"   // DB9
// stored: InstanceOfName DigitalOutput, InstanceOfType FB
"DigitalOutput"
BEGIN
END_DATA_BLOCK

DATA_BLOCK "DoDb"   // DB109
// stored: AutoNumber false, InstanceOfName DoFb, InstanceOfType FB
"DoFb"
BEGIN
END_DATA_BLOCK

DATA_BLOCK "DoFb_DB"   // DB6
// stored: InstanceOfName DoFb, InstanceOfType FB
"DoFb"
BEGIN
END_DATA_BLOCK

DATA_BLOCK "Vessel_Lamp"   // DB1
// stored: AutoNumber false, InstanceOfName TIMER, InstanceOfType FB
"TIMER"
BEGIN
END_DATA_BLOCK
